LIN {X -0.096,Y -433.923,Z 789.927,A 0.000,B 0.000,C 90.000,E1 202.950} C_DIS
LIN {X -0.182,Y -428.835,Z 789.913,A 0.000,B 0.000,C 90.000,E1 200.301} C_DIS
LIN {X -0.108,Y -424.366,Z 789.900,A 0.000,B 0.000,C 90.000,E1 197.946} C_DIS
LIN {X 0.063,Y -420.410,Z 789.888,A 0.000,B 0.000,C 90.000,E1 195.898} C_DIS
LIN {X 0.140,Y -414.585,Z 789.871,A 0.000,B 0.000,C 90.000,E1 192.827} C_DIS
LIN {X -0.010,Y -412.023,Z 789.864,A 0.000,B 0.000,C 90.000,E1 191.478} C_DIS
LIN {X -0.175,Y -407.184,Z 789.849,A 0.000,B 0.000,C 90.000,E1 188.746} C_DIS
LIN {X -0.117,Y -404.851,Z 789.841,A 0.000,B 0.000,C 90.000,E1 187.352} C_DIS
LIN {X 0.135,Y -400.530,Z 789.827,A 0.000,B 0.000,C 90.000,E1 184.878} C_DIS
LIN {X -0.196,Y -393.502,Z 789.800,A 0.000,B 0.000,C 90.000,E1 180.000} C_DIS
LIN {X -0.078,Y -390.107,Z 789.782,A 0.000,B 0.000,C 90.000,E1 176.788} C_DIS
LIN {X -0.091,Y -388.317,Z 789.772,A 0.000,B 0.000,C 90.000,E1 175.008} C_DIS
LIN {X 0.135,Y -385.736,Z 789.758,A 0.000,B 0.000,C 90.000,E1 172.470} C_DIS
LIN {X 0.177,Y -384.408,Z 789.750,A 0.000,B 0.000,C 90.000,E1 171.027} C_DIS
LIN {X -0.013,Y -381.815,Z 789.732,A 0.000,B 0.000,C 90.000,E1 167.813} C_DIS
LIN {X -0.019,Y -380.151,Z 789.718,A 0.000,B 0.000,C 90.000,E1 165.283} C_DIS
LIN {X 0.113,Y -378.893,Z 789.704,A 0.000,B 0.000,C 90.000,E1 162.725} C_DIS
LIN {X 0.069,Y -377.980,Z 789.690,A 0.000,B 0.000,C 90.000,E1 160.188} C_DIS
LIN {X -0.095,Y -377.646,Z 789.676,A 0.000,B 0.000,C 90.000,E1 157.667} C_DIS
LIN {X -0.228,Y -379.156,Z 789.646,A 0.000,B 0.000,C 90.000,E1 152.231} C_DIS
LIN {X 0.139,Y -380.892,Z 789.633,A 0.000,B 0.000,C 90.000,E1 149.999} C_DIS
LIN {X 0.074,Y -383.379,Z 789.623,A 0.000,B 0.000,C 90.000,E1 148.201} C_DIS
LIN {X -0.076,Y -384.604,Z 789.619,A 0.000,B 0.000,C 90.000,E1 147.502} C_DIS
LIN {X 0.144,Y -388.645,Z 789.609,A 0.000,B 0.000,C 90.000,E1 145.674} C_DIS
LIN {X 0.039,Y -390.655,Z 789.606,A 0.000,B 0.000,C 90.000,E1 144.975} C_DIS
LIN {X -0.048,Y -393.112,Z 789.602,A 0.000,B 0.000,C 90.000,E1 144.276} C_DIS
LIN {X 0.119,Y -396.079,Z 789.598,A 0.000,B 0.000,C 90.000,E1 143.543} C_DIS
LIN {X 0.038,Y -400.422,Z 789.593,A 0.000,B 0.000,C 90.000,E1 142.718} C_DIS
LIN {X 0.118,Y -403.485,Z 789.590,A 0.000,B 0.000,C 90.000,E1 142.190} C_DIS
LIN {X 0.232,Y -407.862,Z 789.587,A 0.000,B 0.000,C 90.000,E1 141.537} C_DIS
LIN {X 0.073,Y -425.471,Z 789.574,A 0.000,B 0.000,C 90.000,E1 139.380} C_DIS
LIN {X -0.229,Y -441.850,Z 789.564,A 0.000,B 0.000,C 90.000,E1 137.472} C_DIS
LIN {X -0.276,Y -452.614,Z 789.557,A 0.000,B 0.000,C 90.000,E1 136.215} C_DIS
LIN {X -0.051,Y -461.582,Z 789.550,A 0.000,B 0.000,C 90.000,E1 135.081} C_DIS
LIN {X 0.114,Y -468.893,Z 789.545,A 0.000,B 0.000,C 90.000,E1 134.109} C_DIS
LIN {X 0.245,Y -478.125,Z 789.538,A 0.000,B 0.000,C 90.000,E1 132.852} C_DIS
LIN {X -0.339,Y -485.771,Z 789.532,A 0.000,B 0.000,C 90.000,E1 131.838} C_DIS
LIN {X -0.279,Y -490.960,Z 789.528,A 0.000,B 0.000,C 90.000,E1 131.067} C_DIS
LIN {X 0.220,Y -499.566,Z 789.520,A 0.000,B 0.000,C 90.000,E1 129.644} C_DIS
LIN {X 0.167,Y -505.023,Z 789.515,A 0.000,B 0.000,C 90.000,E1 128.749} C_DIS
LIN {X -0.143,Y -510.126,Z 789.510,A 0.000,B 0.000,C 90.000,E1 127.890} C_DIS
LIN {X -0.009,Y -513.345,Z 789.507,A 0.000,B 0.000,C 90.000,E1 127.282} C_DIS
LIN {X -0.063,Y -520.174,Z 789.500,A 0.000,B 0.000,C 90.000,E1 125.964} C_DIS
LIN {X -0.253,Y -525.997,Z 789.493,A 0.000,B 0.000,C 90.000,E1 124.818} C_DIS
LIN {X 0.086,Y -529.747,Z 789.489,A 0.000,B 0.000,C 90.000,E1 123.913} C_DIS
LIN {X 0.176,Y -533.294,Z 789.484,A 0.000,B 0.000,C 90.000,E1 123.038} C_DIS
LIN {X -0.148,Y -536.722,Z 789.479,A 0.000,B 0.000,C 90.000,E1 122.212} C_DIS
LIN {X 0.021,Y -541.048,Z 789.473,A 0.000,B 0.000,C 90.000,E1 121.052} C_DIS
LIN {X -0.044,Y -544.102,Z 789.468,A 0.000,B 0.000,C 90.000,E1 120.207} C_DIS
LIN {X 0.200,Y -546.907,Z 789.463,A 0.000,B 0.000,C 90.000,E1 119.333} C_DIS
LIN {X -0.036,Y -550.394,Z 789.457,A 0.000,B 0.000,C 90.000,E1 118.231} C_DIS
LIN {X 0.008,Y -552.853,Z 789.452,A 0.000,B 0.000,C 90.000,E1 117.385} C_DIS
LIN {X 0.073,Y -554.977,Z 789.448,A 0.000,B 0.000,C 90.000,E1 116.539} C_DIS
LIN {X -0.087,Y -556.744,Z 789.443,A 0.000,B 0.000,C 90.000,E1 115.720} C_DIS
LIN {X -0.225,Y -558.214,Z 789.438,A 0.000,B 0.000,C 90.000,E1 114.899} C_DIS
LIN {X 0.164,Y -559.424,Z 789.434,A 0.000,B 0.000,C 90.000,E1 114.027} C_DIS
LIN {X 0.157,Y -560.882,Z 789.426,A 0.000,B 0.000,C 90.000,E1 112.642} C_DIS
LIN {X -0.047,Y -562.323,Z 789.418,A 0.000,B 0.000,C 90.000,E1 111.280} C_DIS
LIN {X 0.098,Y -563.529,Z 789.411,A 0.000,B 0.000,C 90.000,E1 109.885} C_DIS
LIN {X -0.262,Y -564.477,Z 789.403,A 0.000,B 0.000,C 90.000,E1 108.544} C_DIS
LIN {X 0.071,Y -565.546,Z 789.394,A 0.000,B 0.000,C 90.000,E1 106.858} C_DIS
LIN {X 0.053,Y -566.949,Z 789.382,A 0.000,B 0.000,C 90.000,E1 104.662} C_DIS
LIN {X -0.061,Y -568.582,Z 789.369,A 0.000,B 0.000,C 90.000,E1 102.479} C_DIS
LIN {X 0.109,Y -570.137,Z 789.359,A 0.000,B 0.000,C 90.000,E1 100.546} C_DIS
LIN {X 0.202,Y -571.656,Z 789.348,A 0.000,B 0.000,C 90.000,E1 98.624} C_DIS
LIN {X -0.147,Y -572.602,Z 789.341,A 0.000,B 0.000,C 90.000,E1 97.296} C_DIS
LIN {X 0.217,Y -573.687,Z 789.331,A 0.000,B 0.000,C 90.000,E1 95.625} C_DIS
LIN {X 0.166,Y -574.755,Z 789.321,A 0.000,B 0.000,C 90.000,E1 93.726} C_DIS
LIN {X -0.229,Y -575.442,Z 789.313,A 0.000,B 0.000,C 90.000,E1 92.407} C_DIS
LIN {X -0.037,Y -575.998,Z 789.306,A 0.000,B 0.000,C 90.000,E1 91.031} C_DIS
LIN {X -0.270,Y -576.652,Z 789.297,A 0.000,B 0.000,C 90.000,E1 89.427} C_DIS
LIN {X 0.193,Y -576.956,Z 789.292,A 0.000,B 0.000,C 90.000,E1 88.568} C_DIS
LIN {X -0.013,Y -577.454,Z 789.283,A 0.000,B 0.000,C 90.000,E1 86.963} C_DIS
LIN {X 0.245,Y -577.727,Z 789.276,A 0.000,B 0.000,C 90.000,E1 85.584} C_DIS
LIN {X 0.144,Y -578.060,Z 789.267,A 0.000,B 0.000,C 90.000,E1 83.970} C_DIS
LIN {X 0.050,Y -578.363,Z 789.258,A 0.000,B 0.000,C 90.000,E1 82.356} C_DIS
LIN {X 0.030,Y -578.620,Z 789.249,A 0.000,B 0.000,C 90.000,E1 80.735} C_DIS
LIN {X 0.107,Y -578.803,Z 789.240,A 0.000,B 0.000,C 90.000,E1 79.106} C_DIS
LIN {X 0.079,Y -578.817,Z 789.232,A 0.000,B 0.000,C 90.000,E1 77.757} C_DIS
LIN {X 0.051,Y -578.707,Z 789.225,A 0.000,B 0.000,C 90.000,E1 76.408} C_DIS
LIN {X -0.061,Y -578.550,Z 789.219,A 0.000,B 0.000,C 90.000,E1 75.338} C_DIS
LIN {X -0.099,Y -578.141,Z 789.208,A 0.000,B 0.000,C 90.000,E1 73.449} C_DIS
LIN {X 0.144,Y -577.788,Z 789.201,A 0.000,B 0.000,C 90.000,E1 72.072} C_DIS
LIN {X -0.007,Y -577.504,Z 789.196,A 0.000,B 0.000,C 90.000,E1 71.275} C_DIS
LIN {X 0.046,Y -576.855,Z 789.187,A 0.000,B 0.000,C 90.000,E1 69.645} C_DIS
LIN {X -0.050,Y -576.024,Z 789.178,A 0.000,B 0.000,C 90.000,E1 68.028} C_DIS
LIN {X 0.008,Y -575.252,Z 789.170,A 0.000,B 0.000,C 90.000,E1 66.666} C_DIS
LIN {X 0.039,Y -574.268,Z 789.163,A 0.000,B 0.000,C 90.000,E1 65.305} C_DIS
LIN {X 0.172,Y -573.461,Z 789.157,A 0.000,B 0.000,C 90.000,E1 64.204} C_DIS
LIN {X -0.113,Y -572.147,Z 789.149,A 0.000,B 0.000,C 90.000,E1 62.871} C_DIS
LIN {X 0.001,Y -570.894,Z 789.143,A 0.000,B 0.000,C 90.000,E1 61.769} C_DIS
LIN {X -0.081,Y -568.995,Z 789.136,A 0.000,B 0.000,C 90.000,E1 60.411} C_DIS
LIN {X -0.047,Y -567.718,Z 789.131,A 0.000,B 0.000,C 90.000,E1 59.587} C_DIS
LIN {X -0.013,Y -565.741,Z 789.125,A 0.000,B 0.000,C 90.000,E1 58.486} C_DIS
LIN {X -0.003,Y -564.109,Z 789.120,A 0.000,B 0.000,C 90.000,E1 57.661} C_DIS
LIN {X -0.005,Y -562.277,Z 789.116,A 0.000,B 0.000,C 90.000,E1 56.834} C_DIS
LIN {X -0.025,Y -560.239,Z 789.111,A 0.000,B 0.000,C 90.000,E1 56.008} C_DIS
LIN {X -0.067,Y -557.981,Z 789.107,A 0.000,B 0.000,C 90.000,E1 55.182} C_DIS
LIN {X -0.137,Y -555.469,Z 789.102,A 0.000,B 0.000,C 90.000,E1 54.356} C_DIS
LIN {X 0.016,Y -553.739,Z 789.099,A 0.000,B 0.000,C 90.000,E1 53.783} C_DIS
LIN {X 0.222,Y -550.798,Z 789.094,A 0.000,B 0.000,C 90.000,E1 52.924} C_DIS
LIN {X -0.038,Y -547.508,Z 789.090,A 0.000,B 0.000,C 90.000,E1 52.110} C_DIS
LIN {X -0.091,Y -544.513,Z 789.086,A 0.000,B 0.000,C 90.000,E1 51.412} C_DIS
LIN {X -0.258,Y -541.278,Z 789.082,A 0.000,B 0.000,C 90.000,E1 50.723} C_DIS
LIN {X 0.130,Y -538.423,Z 789.079,A 0.000,B 0.000,C 90.000,E1 50.114} C_DIS
LIN {X 0.321,Y -534.466,Z 789.075,A 0.000,B 0.000,C 90.000,E1 49.380} C_DIS
LIN {X -0.052,Y -531.062,Z 789.071,A 0.000,B 0.000,C 90.000,E1 48.852} C_DIS
LIN {X 0.254,Y -527.176,Z 789.068,A 0.000,B 0.000,C 90.000,E1 48.243} C_DIS
LIN {X -0.212,Y -522.843,Z 789.065,A 0.000,B 0.000,C 90.000,E1 47.715} C_DIS
LIN {X -0.215,Y -518.175,Z 789.062,A 0.000,B 0.000,C 90.000,E1 47.148} C_DIS
LIN {X -0.127,Y -514.389,Z 789.059,A 0.000,B 0.000,C 90.000,E1 46.701} C_DIS
LIN {X -0.219,Y -508.950,Z 789.056,A 0.000,B 0.000,C 90.000,E1 46.134} C_DIS
LIN {X -0.306,Y -504.703,Z 789.054,A 0.000,B 0.000,C 90.000,E1 45.729} C_DIS
LIN {X -0.045,Y -497.382,Z 789.050,A 0.000,B 0.000,C 90.000,E1 45.040} C_DIS
LIN {X 0.203,Y -494.493,Z 789.049,A 0.000,B 0.000,C 90.000,E1 44.757} C_DIS
LIN {X -0.244,Y -486.605,Z 789.045,A 0.000,B 0.000,C 90.000,E1 44.190} C_DIS
LIN {X -0.048,Y -478.786,Z 789.042,A 0.000,B 0.000,C 90.000,E1 43.581} C_DIS
LIN {X -0.066,Y -465.969,Z 789.037,A 0.000,B 0.000,C 90.000,E1 42.690} C_DIS
LIN {X -0.267,Y -452.980,Z 789.032,A 0.000,B 0.000,C 90.000,E1 41.838} C_DIS
LIN {X -0.082,Y -427.596,Z 789.022,A 0.000,B 0.000,C 90.000,E1 40.011} C_DIS
LIN {X -0.153,Y -415.102,Z 789.017,A 0.000,B 0.000,C 90.000,E1 39.036} C_DIS
LIN {X -0.015,Y -409.294,Z 789.014,A 0.000,B 0.000,C 90.000,E1 38.508} C_DIS
LIN {X -0.120,Y -404.958,Z 789.012,A 0.000,B 0.000,C 90.000,E1 38.096} C_DIS
LIN {X -0.153,Y -404.943,Z 789.012,A 0.000,B 0.000,C 90.000,E1 38.096} C_DIS
LIN {X -0.008,Y -396.699,Z 788.988,A 0.000,B 0.000,C 90.000,E1 33.785} C_DIS
LIN {X 0.077,Y -395.965,Z 788.985,A 0.000,B 0.000,C 90.000,E1 33.245} C_DIS
LIN {X 0.145,Y -396.699,Z 788.970,A 0.000,B 0.000,C 90.000,E1 30.590} C_DIS
LIN {X 0.174,Y -398.039,Z 788.954,A 0.000,B 0.000,C 90.000,E1 27.769} C_DIS
LIN {X -0.003,Y -399.440,Z 788.941,A 0.000,B 0.000,C 90.000,E1 25.335} C_DIS
LIN {X 0.178,Y -400.863,Z 788.929,A 0.000,B 0.000,C 90.000,E1 23.206} C_DIS
LIN {X 0.143,Y -403.490,Z 788.912,A 0.000,B 0.000,C 90.000,E1 20.066} C_DIS
LIN {X 0.024,Y -407.875,Z 788.890,A 0.000,B 0.000,C 90.000,E1 16.260} C_DIS
LIN {X -0.123,Y -412.436,Z 788.873,A 0.000,B 0.000,C 90.000,E1 13.175} C_DIS
LIN {X -0.165,Y -416.506,Z 788.860,A 0.000,B 0.000,C 90.000,E1 10.782} C_DIS
LIN {X -0.227,Y -420.048,Z 788.848,A 0.000,B 0.000,C 90.000,E1 8.746} C_DIS
LIN {X 0.150,Y -423.655,Z 788.837,A 0.000,B 0.000,C 90.000,E1 6.663} C_DIS
LIN {X 0.189,Y -427.918,Z 788.824,A 0.000,B 0.000,C 90.000,E1 4.302} C_DIS
LIN {X 0.210,Y -431.687,Z 788.813,A 0.000,B 0.000,C 90.000,E1 2.293} C_DIS
LIN {X 0.165,Y -436.770,Z 788.799,A 0.000,B 0.000,C 90.000,E1 359.771} C_DIS
LIN {X 0.176,Y -442.483,Z 788.784,A 0.000,B 0.000,C 90.000,E1 357.135} C_DIS
LIN {X -0.176,Y -447.843,Z 788.772,A 0.000,B 0.000,C 90.000,E1 354.894} C_DIS
LIN {X 0.104,Y -453.252,Z 788.759,A 0.000,B 0.000,C 90.000,E1 352.591} C_DIS
LIN {X 0.199,Y -457.058,Z 788.750,A 0.000,B 0.000,C 90.000,E1 350.971} C_DIS
LIN {X -0.188,Y -463.295,Z 788.736,A 0.000,B 0.000,C 90.000,E1 348.465} C_DIS
LIN {X -0.048,Y -465.363,Z 788.732,A 0.000,B 0.000,C 90.000,E1 347.813} C_DIS
LIN {X 0.209,Y -466.568,Z 788.731,A 0.000,B 0.000,C 90.000,E1 347.465} C_DIS
LIN {X -0.121,Y -468.502,Z 788.728,A 0.000,B 0.000,C 90.000,E1 347.117} C_DIS
LIN {X 0.118,Y -471.921,Z 788.726,A 0.000,B 0.000,C 90.000,E1 346.589} C_DIS
LIN {X 0.192,Y -476.026,Z 788.723,A 0.000,B 0.000,C 90.000,E1 346.117} C_DIS
LIN {X 0.085,Y -481.163,Z 788.720,A 0.000,B 0.000,C 90.000,E1 345.644} C_DIS
LIN {X 0.074,Y -492.813,Z 788.715,A 0.000,B 0.000,C 90.000,E1 344.755} C_DIS
LIN {X -0.016,Y -511.779,Z 788.708,A 0.000,B 0.000,C 90.000,E1 343.449} C_DIS
LIN {X -0.203,Y -530.426,Z 788.701,A 0.000,B 0.000,C 90.000,E1 342.236} C_DIS
LIN {X 0.002,Y -538.135,Z 788.698,A 0.000,B 0.000,C 90.000,E1 341.692} C_DIS
LIN {X -0.207,Y -548.725,Z 788.694,A 0.000,B 0.000,C 90.000,E1 340.967} C_DIS
LIN {X 0.155,Y -555.920,Z 788.691,A 0.000,B 0.000,C 90.000,E1 340.369} C_DIS
LIN {X 0.240,Y -561.405,Z 788.688,A 0.000,B 0.000,C 90.000,E1 339.880} C_DIS
LIN {X 0.036,Y -566.649,Z 788.686,A 0.000,B 0.000,C 90.000,E1 339.390} C_DIS
LIN {X 0.117,Y -571.621,Z 788.683,A 0.000,B 0.000,C 90.000,E1 338.847} C_DIS
LIN {X 0.246,Y -577.291,Z 788.679,A 0.000,B 0.000,C 90.000,E1 338.156} C_DIS
LIN {X 0.113,Y -583.671,Z 788.674,A 0.000,B 0.000,C 90.000,E1 337.358} C_DIS
LIN {X 0.330,Y -588.579,Z 788.671,A 0.000,B 0.000,C 90.000,E1 336.666} C_DIS
LIN {X 0.206,Y -595.966,Z 788.665,A 0.000,B 0.000,C 90.000,E1 335.613} C_DIS
LIN {X -0.085,Y -602.129,Z 788.660,A 0.000,B 0.000,C 90.000,E1 334.717} C_DIS
LIN {X 0.220,Y -608.704,Z 788.654,A 0.000,B 0.000,C 90.000,E1 333.640} C_DIS
LIN {X 0.067,Y -614.861,Z 788.648,A 0.000,B 0.000,C 90.000,E1 332.615} C_DIS
LIN {X -0.004,Y -620.008,Z 788.643,A 0.000,B 0.000,C 90.000,E1 331.719} C_DIS
LIN {X -0.264,Y -625.689,Z 788.637,A 0.000,B 0.000,C 90.000,E1 330.717} C_DIS
LIN {X 0.103,Y -631.070,Z 788.632,A 0.000,B 0.000,C 90.000,E1 329.665} C_DIS
LIN {X 0.016,Y -636.701,Z 788.625,A 0.000,B 0.000,C 90.000,E1 328.535} C_DIS
LIN {X -0.071,Y -640.189,Z 788.621,A 0.000,B 0.000,C 90.000,E1 327.788} C_DIS
LIN {X -0.073,Y -644.643,Z 788.615,A 0.000,B 0.000,C 90.000,E1 326.786} C_DIS
LIN {X -0.147,Y -646.699,Z 788.613,A 0.000,B 0.000,C 90.000,E1 326.294} C_DIS
LIN {X -0.246,Y -650.752,Z 788.607,A 0.000,B 0.000,C 90.000,E1 325.308} C_DIS
LIN {X 0.245,Y -654.480,Z 788.602,A 0.000,B 0.000,C 90.000,E1 324.276} C_DIS
LIN {X -0.280,Y -658.009,Z 788.596,A 0.000,B 0.000,C 90.000,E1 323.336} C_DIS
LIN {X -0.278,Y -662.012,Z 788.589,A 0.000,B 0.000,C 90.000,E1 322.110} C_DIS
LIN {X -0.214,Y -665.758,Z 788.583,A 0.000,B 0.000,C 90.000,E1 320.884} C_DIS
LIN {X -0.185,Y -669.185,Z 788.576,A 0.000,B 0.000,C 90.000,E1 319.666} C_DIS
LIN {X -0.102,Y -671.762,Z 788.570,A 0.000,B 0.000,C 90.000,E1 318.690} C_DIS
LIN {X 0.027,Y -674.793,Z 788.564,A 0.000,B 0.000,C 90.000,E1 317.472} C_DIS
LIN {X -0.298,Y -677.372,Z 788.557,A 0.000,B 0.000,C 90.000,E1 316.296} C_DIS
LIN {X -0.026,Y -680.472,Z 788.548,A 0.000,B 0.000,C 90.000,E1 314.595} C_DIS
LIN {X 0.209,Y -682.391,Z 788.541,A 0.000,B 0.000,C 90.000,E1 313.380} C_DIS
LIN {X -0.001,Y -684.231,Z 788.535,A 0.000,B 0.000,C 90.000,E1 312.204} C_DIS
LIN {X 0.327,Y -685.870,Z 788.528,A 0.000,B 0.000,C 90.000,E1 310.987} C_DIS
LIN {X 0.239,Y -687.268,Z 788.521,A 0.000,B 0.000,C 90.000,E1 309.806} C_DIS
LIN {X 0.180,Y -688.502,Z 788.515,A 0.000,B 0.000,C 90.000,E1 308.624} C_DIS
LIN {X -0.186,Y -690.165,Z 788.505,A 0.000,B 0.000,C 90.000,E1 306.996} C_DIS
LIN {X -0.438,Y -691.394,Z 788.498,A 0.000,B 0.000,C 90.000,E1 305.598} C_DIS
LIN {X -0.302,Y -692.289,Z 788.491,A 0.000,B 0.000,C 90.000,E1 304.405} C_DIS
LIN {X -0.290,Y -693.500,Z 788.482,A 0.000,B 0.000,C 90.000,E1 302.752} C_DIS
LIN {X -0.032,Y -694.830,Z 788.473,A 0.000,B 0.000,C 90.000,E1 301.082} C_DIS
LIN {X 0.111,Y -695.492,Z 788.467,A 0.000,B 0.000,C 90.000,E1 300.129} C_DIS
LIN {X -0.197,Y -696.213,Z 788.460,A 0.000,B 0.000,C 90.000,E1 298.743} C_DIS
LIN {X 0.215,Y -696.715,Z 788.454,A 0.000,B 0.000,C 90.000,E1 297.769} C_DIS
LIN {X 0.216,Y -697.495,Z 788.447,A 0.000,B 0.000,C 90.000,E1 296.360} C_DIS
LIN {X 0.232,Y -698.424,Z 788.439,A 0.000,B 0.000,C 90.000,E1 294.951} C_DIS
LIN {X -0.169,Y -698.589,Z 788.436,A 0.000,B 0.000,C 90.000,E1 294.515} C_DIS
LIN {X 0.094,Y -698.627,Z 788.435,A 0.000,B 0.000,C 90.000,E1 294.259} C_DIS
LIN {X 0.072,Y -698.429,Z 788.434,A 0.000,B 0.000,C 90.000,E1 294.027} C_DIS
LIN {X -0.042,Y -697.521,Z 788.431,A 0.000,B 0.000,C 90.000,E1 293.567} C_DIS
LIN {X -0.060,Y -696.532,Z 788.430,A 0.000,B 0.000,C 90.000,E1 293.334} C_DIS
LIN {X 0.321,Y -693.962,Z 788.428,A 0.000,B 0.000,C 90.000,E1 292.950} C_DIS
LIN {X -0.341,Y -692.008,Z 788.426,A 0.000,B 0.000,C 90.000,E1 292.770} C_DIS
LIN {X -0.220,Y -690.406,Z 788.426,A 0.000,B 0.000,C 90.000,E1 292.642} C_DIS
LIN {X 0.151,Y -686.156,Z 788.425,A 0.000,B 0.000,C 90.000,E1 292.408} C_DIS
LIN {X -0.086,Y -682.793,Z 788.424,A 0.000,B 0.000,C 90.000,E1 292.280} C_DIS
LIN {X -0.037,Y -680.715,Z 788.423,A 0.000,B 0.000,C 90.000,E1 292.206} C_DIS
LIN {X 0.087,Y -674.471,Z 788.422,A 0.000,B 0.000,C 90.000,E1 292.025} C_DIS
LIN {X -0.131,Y -669.195,Z 788.422,A 0.000,B 0.000,C 90.000,E1 291.950} C_DIS
LIN {X -0.150,Y -651.406,Z 788.420,A 0.000,B 0.000,C 90.000,E1 291.663} C_DIS
LIN {X -0.111,Y -634.211,Z 788.419,A 0.000,B 0.000,C 90.000,E1 291.334} C_DIS
LIN {X -0.087,Y -613.288,Z 788.416,A 0.000,B 0.000,C 90.000,E1 290.865} C_DIS
LIN {X -0.083,Y -596.538,Z 788.414,A 0.000,B 0.000,C 90.000,E1 290.429} C_DIS
LIN {X 0.072,Y -586.447,Z 788.412,A 0.000,B 0.000,C 90.000,E1 290.120} C_DIS
LIN {X -0.132,Y -576.325,Z 788.410,A 0.000,B 0.000,C 90.000,E1 289.812} C_DIS
LIN {X -0.045,Y -569.864,Z 788.409,A 0.000,B 0.000,C 90.000,E1 289.577} C_DIS
LIN {X 0.055,Y -564.207,Z 788.407,A 0.000,B 0.000,C 90.000,E1 289.322} C_DIS
LIN {X 0.105,Y -562.387,Z 788.407,A 0.000,B 0.000,C 90.000,E1 289.214} C_DIS
LIN {X -0.020,Y -558.873,Z 788.405,A 0.000,B 0.000,C 90.000,E1 288.960} C_DIS
LIN {X -0.139,Y -557.615,Z 788.404,A 0.000,B 0.000,C 90.000,E1 288.779} C_DIS
LIN {X 0.273,Y -556.882,Z 788.404,A 0.000,B 0.000,C 90.000,E1 288.598} C_DIS
LIN {X 0.139,Y -555.816,Z 788.402,A 0.000,B 0.000,C 90.000,E1 288.308} C_DIS
LIN {X -0.011,Y -555.004,Z 788.400,A 0.000,B 0.000,C 90.000,E1 287.946} C_DIS
LIN {X -0.143,Y -554.325,Z 788.397,A 0.000,B 0.000,C 90.000,E1 287.402} C_DIS
LIN {X -0.156,Y -552.737,Z 788.376,A 0.000,B 0.000,C 90.000,E1 283.772} C_DIS
LIN {X 0.147,Y -552.218,Z 788.367,A 0.000,B 0.000,C 90.000,E1 282.063} C_DIS
LIN {X -0.210,Y -551.653,Z 788.356,A 0.000,B 0.000,C 90.000,E1 280.141} C_DIS
LIN {X 0.104,Y -551.022,Z 788.342,A 0.000,B 0.000,C 90.000,E1 277.587} C_DIS
LIN {X -0.085,Y -550.591,Z 788.336,A 0.000,B 0.000,C 90.000,E1 276.486} C_DIS
LIN {X -0.213,Y -549.742,Z 788.327,A 0.000,B 0.000,C 90.000,E1 274.816} C_DIS
LIN {X 0.062,Y -548.791,Z 788.319,A 0.000,B 0.000,C 90.000,E1 273.383} C_DIS
LIN {X -0.104,Y -547.554,Z 788.308,A 0.000,B 0.000,C 90.000,E1 271.432} C_DIS
LIN {X 0.170,Y -546.472,Z 788.299,A 0.000,B 0.000,C 90.000,E1 269.714} C_DIS
LIN {X -0.168,Y -545.463,Z 788.291,A 0.000,B 0.000,C 90.000,E1 268.339} C_DIS
LIN {X 0.094,Y -544.340,Z 788.281,A 0.000,B 0.000,C 90.000,E1 266.617} C_DIS
LIN {X -0.272,Y -543.516,Z 788.273,A 0.000,B 0.000,C 90.000,E1 265.241} C_DIS
LIN {X -0.009,Y -542.383,Z 788.264,A 0.000,B 0.000,C 90.000,E1 263.514} C_DIS
LIN {X 0.293,Y -541.219,Z 788.256,A 0.000,B 0.000,C 90.000,E1 262.064} C_DIS
LIN {X 0.109,Y -539.568,Z 788.245,A 0.000,B 0.000,C 90.000,E1 260.095} C_DIS
LIN {X -0.237,Y -538.504,Z 788.239,A 0.000,B 0.000,C 90.000,E1 258.993} C_DIS
LIN {X 0.266,Y -536.864,Z 788.229,A 0.000,B 0.000,C 90.000,E1 257.229} C_DIS
LIN {X -0.019,Y -535.770,Z 788.223,A 0.000,B 0.000,C 90.000,E1 256.117} C_DIS
LIN {X 0.081,Y -533.559,Z 788.212,A 0.000,B 0.000,C 90.000,E1 254.102} C_DIS
LIN {X 0.239,Y -531.630,Z 788.202,A 0.000,B 0.000,C 90.000,E1 252.362} C_DIS
LIN {X -0.166,Y -529.904,Z 788.194,A 0.000,B 0.000,C 90.000,E1 250.967} C_DIS
LIN {X 0.076,Y -527.478,Z 788.185,A 0.000,B 0.000,C 90.000,E1 249.209} C_DIS
LIN {X -0.220,Y -525.416,Z 788.177,A 0.000,B 0.000,C 90.000,E1 247.794} C_DIS
LIN {X -0.035,Y -523.614,Z 788.170,A 0.000,B 0.000,C 90.000,E1 246.613} C_DIS
LIN {X 0.017,Y -521.396,Z 788.162,A 0.000,B 0.000,C 90.000,E1 245.153} C_DIS
LIN {X 0.035,Y -519.030,Z 788.154,A 0.000,B 0.000,C 90.000,E1 243.691} C_DIS
LIN {X -0.124,Y -517.079,Z 788.147,A 0.000,B 0.000,C 90.000,E1 242.538} C_DIS
LIN {X 0.023,Y -515.509,Z 788.143,A 0.000,B 0.000,C 90.000,E1 241.641} C_DIS
LIN {X -0.298,Y -512.749,Z 788.134,A 0.000,B 0.000,C 90.000,E1 240.205} C_DIS
LIN {X 0.285,Y -509.978,Z 788.126,A 0.000,B 0.000,C 90.000,E1 238.663} C_DIS
LIN {X 0.004,Y -506.328,Z 788.116,A 0.000,B 0.000,C 90.000,E1 236.914} C_DIS
LIN {X 0.109,Y -504.427,Z 788.111,A 0.000,B 0.000,C 90.000,E1 236.008} C_DIS
LIN {X 0.083,Y -501.692,Z 788.105,A 0.000,B 0.000,C 90.000,E1 234.815} C_DIS
LIN {X 0.139,Y -499.536,Z 788.100,A 0.000,B 0.000,C 90.000,E1 233.909} C_DIS
LIN {X -0.100,Y -495.775,Z 788.091,A 0.000,B 0.000,C 90.000,E1 232.431} C_DIS
LIN {X 0.199,Y -490.501,Z 788.079,A 0.000,B 0.000,C 90.000,E1 230.275} C_DIS
LIN {X -0.046,Y -484.219,Z 788.064,A 0.000,B 0.000,C 90.000,E1 227.553} C_DIS
LIN {X -0.248,Y -480.260,Z 788.054,A 0.000,B 0.000,C 90.000,E1 225.729} C_DIS
LIN {X -0.315,Y -476.825,Z 788.045,A 0.000,B 0.000,C 90.000,E1 224.190} C_DIS
LIN {X -0.108,Y -473.429,Z 788.037,A 0.000,B 0.000,C 90.000,E1 222.609} C_DIS
LIN {X -0.011,Y -468.094,Z 788.023,A 0.000,B 0.000,C 90.000,E1 220.092} C_DIS
LIN {X 0.175,Y -464.060,Z 788.012,A 0.000,B 0.000,C 90.000,E1 218.177} C_DIS
LIN {X -0.159,Y -461.517,Z 788.005,A 0.000,B 0.000,C 90.000,E1 216.950} C_DIS
LIN {X 0.066,Y -456.774,Z 787.993,A 0.000,B 0.000,C 90.000,E1 214.692} C_DIS
LIN {X 0.181,Y -452.912,Z 787.982,A 0.000,B 0.000,C 90.000,E1 212.752} C_DIS
LIN {X -0.199,Y -448.467,Z 787.970,A 0.000,B 0.000,C 90.000,E1 210.541} C_DIS
LIN {X 0.015,Y -444.689,Z 787.959,A 0.000,B 0.000,C 90.000,E1 208.565} C_DIS
LIN {X 0.079,Y -441.606,Z 787.950,A 0.000,B 0.000,C 90.000,E1 206.924} C_DIS
LIN {X 0.075,Y -438.468,Z 787.941,A 0.000,B 0.000,C 90.000,E1 205.283} C_DIS
LIN {X -0.154,Y -434.747,Z 787.930,A 0.000,B 0.000,C 90.000,E1 203.334} C_DIS
LIN {X -0.053,Y -429.614,Z 787.915,A 0.000,B 0.000,C 90.000,E1 200.663} C_DIS
LIN {X -0.022,Y -427.031,Z 787.907,A 0.000,B 0.000,C 90.000,E1 199.322} C_DIS
LIN {X 0.023,Y -423.876,Z 787.898,A 0.000,B 0.000,C 90.000,E1 197.638} C_DIS
LIN {X -0.112,Y -420.584,Z 787.889,A 0.000,B 0.000,C 90.000,E1 195.969} C_DIS
LIN {X 0.081,Y -414.772,Z 787.872,A 0.000,B 0.000,C 90.000,E1 192.883} C_DIS
LIN {X -0.106,Y -412.860,Z 787.866,A 0.000,B 0.000,C 90.000,E1 191.883} C_DIS
LIN {X -0.196,Y -406.222,Z 787.845,A 0.000,B 0.000,C 90.000,E1 188.106} C_DIS
LIN {X -0.209,Y -403.792,Z 787.837,A 0.000,B 0.000,C 90.000,E1 186.720} C_DIS
LIN {X 0.070,Y -400.201,Z 787.826,A 0.000,B 0.000,C 90.000,E1 184.588} C_DIS
LIN {X 0.160,Y -393.706,Z 787.800,A 0.000,B 0.000,C 90.000,E1 180.000} C_DIS
LIN {X -0.108,Y -390.325,Z 787.782,A 0.000,B 0.000,C 90.000,E1 176.846} C_DIS
LIN {X -0.116,Y -388.547,Z 787.773,A 0.000,B 0.000,C 90.000,E1 175.065} C_DIS
LIN {X -0.129,Y -386.637,Z 787.763,A 0.000,B 0.000,C 90.000,E1 173.280} C_DIS
LIN {X -0.141,Y -385.015,Z 787.753,A 0.000,B 0.000,C 90.000,E1 171.489} C_DIS
LIN {X -0.005,Y -382.332,Z 787.735,A 0.000,B 0.000,C 90.000,E1 168.229} C_DIS
LIN {X 0.100,Y -381.303,Z 787.727,A 0.000,B 0.000,C 90.000,E1 166.769} C_DIS
LIN {X -0.003,Y -380.492,Z 787.719,A 0.000,B 0.000,C 90.000,E1 165.338} C_DIS
LIN {X 0.141,Y -379.058,Z 787.702,A 0.000,B 0.000,C 90.000,E1 162.417} C_DIS
LIN {X 0.113,Y -378.334,Z 787.690,A 0.000,B 0.000,C 90.000,E1 160.242} C_DIS
LIN {X -0.050,Y -377.905,Z 787.674,A 0.000,B 0.000,C 90.000,E1 157.358} C_DIS
LIN {X 0.098,Y -380.351,Z 787.638,A 0.000,B 0.000,C 90.000,E1 150.795} C_DIS
LIN {X -0.135,Y -381.354,Z 787.632,A 0.000,B 0.000,C 90.000,E1 149.744} C_DIS
LIN {X 0.007,Y -383.825,Z 787.622,A 0.000,B 0.000,C 90.000,E1 147.916} C_DIS
LIN {X 0.015,Y -385.857,Z 787.616,A 0.000,B 0.000,C 90.000,E1 146.834} C_DIS
LIN {X 0.041,Y -388.165,Z 787.610,A 0.000,B 0.000,C 90.000,E1 145.754} C_DIS
LIN {X -0.069,Y -390.042,Z 787.606,A 0.000,B 0.000,C 90.000,E1 145.055} C_DIS
LIN {X 0.030,Y -392.955,Z 787.601,A 0.000,B 0.000,C 90.000,E1 144.149} C_DIS
LIN {X 0.194,Y -395.894,Z 787.597,A 0.000,B 0.000,C 90.000,E1 143.417} C_DIS
LIN {X 0.049,Y -397.657,Z 787.595,A 0.000,B 0.000,C 90.000,E1 143.084} C_DIS
LIN {X -0.170,Y -399.340,Z 787.593,A 0.000,B 0.000,C 90.000,E1 142.763} C_DIS
LIN {X 0.154,Y -402.307,Z 787.590,A 0.000,B 0.000,C 90.000,E1 142.190} C_DIS
LIN {X -0.178,Y -406.358,Z 787.587,A 0.000,B 0.000,C 90.000,E1 141.618} C_DIS
LIN {X 0.056,Y -412.295,Z 787.582,A 0.000,B 0.000,C 90.000,E1 140.803} C_DIS
LIN {X 0.126,Y -427.124,Z 787.572,A 0.000,B 0.000,C 90.000,E1 139.013} C_DIS
LIN {X -0.218,Y -440.692,Z 787.564,A 0.000,B 0.000,C 90.000,E1 137.472} C_DIS
LIN {X 0.253,Y -452.471,Z 787.556,A 0.000,B 0.000,C 90.000,E1 136.053} C_DIS
LIN {X -0.120,Y -460.214,Z 787.551,A 0.000,B 0.000,C 90.000,E1 135.162} C_DIS
LIN {X -0.030,Y -466.152,Z 787.547,A 0.000,B 0.000,C 90.000,E1 134.393} C_DIS
LIN {X -0.143,Y -473.272,Z 787.541,A 0.000,B 0.000,C 90.000,E1 133.461} C_DIS
LIN {X -0.212,Y -477.920,Z 787.538,A 0.000,B 0.000,C 90.000,E1 132.852} C_DIS
LIN {X -0.090,Y -485.608,Z 787.532,A 0.000,B 0.000,C 90.000,E1 131.757} C_DIS
LIN {X -0.131,Y -489.877,Z 787.529,A 0.000,B 0.000,C 90.000,E1 131.148} C_DIS
LIN {X -0.122,Y -497.694,Z 787.522,A 0.000,B 0.000,C 90.000,E1 129.930} C_DIS
LIN {X 0.191,Y -503.220,Z 787.517,A 0.000,B 0.000,C 90.000,E1 128.991} C_DIS
LIN {X -0.028,Y -509.343,Z 787.511,A 0.000,B 0.000,C 90.000,E1 127.971} C_DIS
LIN {X -0.093,Y -513.362,Z 787.507,A 0.000,B 0.000,C 90.000,E1 127.237} C_DIS
LIN {X 0.164,Y -520.220,Z 787.500,A 0.000,B 0.000,C 90.000,E1 125.884} C_DIS
LIN {X -0.025,Y -526.077,Z 787.493,A 0.000,B 0.000,C 90.000,E1 124.739} C_DIS
LIN {X -0.068,Y -531.614,Z 787.486,A 0.000,B 0.000,C 90.000,E1 123.452} C_DIS
LIN {X 0.183,Y -535.684,Z 787.480,A 0.000,B 0.000,C 90.000,E1 122.418} C_DIS
LIN {X -0.119,Y -538.982,Z 787.475,A 0.000,B 0.000,C 90.000,E1 121.592} C_DIS
LIN {X 0.069,Y -542.119,Z 787.471,A 0.000,B 0.000,C 90.000,E1 120.718} C_DIS
LIN {X 0.018,Y -545.082,Z 787.466,A 0.000,B 0.000,C 90.000,E1 119.873} C_DIS
LIN {X 0.005,Y -547.844,Z 787.461,A 0.000,B 0.000,C 90.000,E1 119.027} C_DIS
LIN {X 0.024,Y -550.471,Z 787.457,A 0.000,B 0.000,C 90.000,E1 118.180} C_DIS
LIN {X 0.072,Y -552.936,Z 787.452,A 0.000,B 0.000,C 90.000,E1 117.334} C_DIS
LIN {X 0.142,Y -555.067,Z 787.447,A 0.000,B 0.000,C 90.000,E1 116.488} C_DIS
LIN {X -0.013,Y -556.853,Z 787.443,A 0.000,B 0.000,C 90.000,E1 115.668} C_DIS
LIN {X 0.088,Y -558.319,Z 787.438,A 0.000,B 0.000,C 90.000,E1 114.823} C_DIS
LIN {X -0.036,Y -559.497,Z 787.433,A 0.000,B 0.000,C 90.000,E1 114.003} C_DIS
LIN {X -0.270,Y -560.955,Z 787.426,A 0.000,B 0.000,C 90.000,E1 112.642} C_DIS
LIN {X 0.050,Y -562.425,Z 787.418,A 0.000,B 0.000,C 90.000,E1 111.227} C_DIS
LIN {X -0.136,Y -563.637,Z 787.410,A 0.000,B 0.000,C 90.000,E1 109.866} C_DIS
LIN {X -0.152,Y -564.633,Z 787.403,A 0.000,B 0.000,C 90.000,E1 108.489} C_DIS
LIN {X 0.190,Y -565.735,Z 787.393,A 0.000,B 0.000,C 90.000,E1 106.804} C_DIS
LIN {X 0.327,Y -567.191,Z 787.381,A 0.000,B 0.000,C 90.000,E1 104.592} C_DIS
LIN {X 0.205,Y -568.889,Z 787.369,A 0.000,B 0.000,C 90.000,E1 102.411} C_DIS
LIN {X -0.295,Y -570.447,Z 787.358,A 0.000,B 0.000,C 90.000,E1 100.546} C_DIS
LIN {X -0.196,Y -571.989,Z 787.348,A 0.000,B 0.000,C 90.000,E1 98.624} C_DIS
LIN {X -0.162,Y -572.765,Z 787.342,A 0.000,B 0.000,C 90.000,E1 97.530} C_DIS
LIN {X 0.272,Y -573.857,Z 787.333,A 0.000,B 0.000,C 90.000,E1 95.853} C_DIS
LIN {X -0.101,Y -574.615,Z 787.325,A 0.000,B 0.000,C 90.000,E1 94.531} C_DIS
LIN {X 0.076,Y -575.392,Z 787.318,A 0.000,B 0.000,C 90.000,E1 93.154} C_DIS
LIN {X 0.293,Y -576.046,Z 787.310,A 0.000,B 0.000,C 90.000,E1 91.776} C_DIS
LIN {X -0.097,Y -576.590,Z 787.303,A 0.000,B 0.000,C 90.000,E1 90.458} C_DIS
LIN {X 0.259,Y -577.277,Z 787.294,A 0.000,B 0.000,C 90.000,E1 88.797} C_DIS
LIN {X -0.095,Y -577.661,Z 787.286,A 0.000,B 0.000,C 90.000,E1 87.478} C_DIS
LIN {X 0.134,Y -578.029,Z 787.278,A 0.000,B 0.000,C 90.000,E1 86.102} C_DIS
LIN {X 0.032,Y -578.342,Z 787.269,A 0.000,B 0.000,C 90.000,E1 84.489} C_DIS
LIN {X -0.054,Y -578.652,Z 787.260,A 0.000,B 0.000,C 90.000,E1 82.875} C_DIS
LIN {X -0.281,Y -578.867,Z 787.253,A 0.000,B 0.000,C 90.000,E1 81.546} C_DIS
LIN {X -0.067,Y -579.000,Z 787.247,A 0.000,B 0.000,C 90.000,E1 80.443} C_DIS
LIN {X -0.202,Y -579.144,Z 787.239,A 0.000,B 0.000,C 90.000,E1 79.106} C_DIS
LIN {X 0.119,Y -579.149,Z 787.233,A 0.000,B 0.000,C 90.000,E1 77.993} C_DIS
LIN {X 0.096,Y -579.046,Z 787.226,A 0.000,B 0.000,C 90.000,E1 76.645} C_DIS
LIN {X 0.206,Y -578.834,Z 787.218,A 0.000,B 0.000,C 90.000,E1 75.283} C_DIS
LIN {X 0.334,Y -578.399,Z 787.208,A 0.000,B 0.000,C 90.000,E1 73.378} C_DIS
LIN {X 0.213,Y -578.093,Z 787.202,A 0.000,B 0.000,C 90.000,E1 72.308} C_DIS
LIN {X 0.067,Y -577.871,Z 787.197,A 0.000,B 0.000,C 90.000,E1 71.511} C_DIS
LIN {X -0.028,Y -577.050,Z 787.187,A 0.000,B 0.000,C 90.000,E1 69.625} C_DIS
LIN {X 0.213,Y -576.188,Z 787.178,A 0.000,B 0.000,C 90.000,E1 67.975} C_DIS
LIN {X 0.268,Y -575.380,Z 787.170,A 0.000,B 0.000,C 90.000,E1 66.613} C_DIS
LIN {X 0.014,Y -574.369,Z 787.163,A 0.000,B 0.000,C 90.000,E1 65.281} C_DIS
LIN {X -0.092,Y -573.542,Z 787.157,A 0.000,B 0.000,C 90.000,E1 64.204} C_DIS
LIN {X 0.134,Y -572.180,Z 787.149,A 0.000,B 0.000,C 90.000,E1 62.820} C_DIS
LIN {X -0.260,Y -570.873,Z 787.143,A 0.000,B 0.000,C 90.000,E1 61.769} C_DIS
LIN {X -0.060,Y -568.939,Z 787.135,A 0.000,B 0.000,C 90.000,E1 60.383} C_DIS
LIN {X 0.183,Y -567.631,Z 787.131,A 0.000,B 0.000,C 90.000,E1 59.537} C_DIS
LIN {X 0.021,Y -565.593,Z 787.125,A 0.000,B 0.000,C 90.000,E1 58.456} C_DIS
LIN {X -0.265,Y -563.925,Z 787.120,A 0.000,B 0.000,C 90.000,E1 57.661} C_DIS
LIN {X -0.268,Y -562.039,Z 787.116,A 0.000,B 0.000,C 90.000,E1 56.834} C_DIS
LIN {X 0.175,Y -559.940,Z 787.111,A 0.000,B 0.000,C 90.000,E1 55.960} C_DIS
LIN {X -0.333,Y -557.635,Z 787.106,A 0.000,B 0.000,C 90.000,E1 55.182} C_DIS
LIN {X -0.003,Y -554.160,Z 787.100,A 0.000,B 0.000,C 90.000,E1 54.036} C_DIS
LIN {X -0.183,Y -552.295,Z 787.097,A 0.000,B 0.000,C 90.000,E1 53.497} C_DIS
LIN {X -0.051,Y -550.298,Z 787.094,A 0.000,B 0.000,C 90.000,E1 52.924} C_DIS
LIN {X 0.116,Y -546.898,Z 787.089,A 0.000,B 0.000,C 90.000,E1 52.065} C_DIS
LIN {X -0.032,Y -543.835,Z 787.085,A 0.000,B 0.000,C 90.000,E1 51.376} C_DIS
LIN {X 0.217,Y -540.506,Z 787.082,A 0.000,B 0.000,C 90.000,E1 50.642} C_DIS
LIN {X -0.161,Y -537.590,Z 787.078,A 0.000,B 0.000,C 90.000,E1 50.114} C_DIS
LIN {X -0.146,Y -534.414,Z 787.075,A 0.000,B 0.000,C 90.000,E1 49.542} C_DIS
LIN {X 0.187,Y -530.918,Z 787.072,A 0.000,B 0.000,C 90.000,E1 48.933} C_DIS
LIN {X -0.255,Y -527.009,Z 787.069,A 0.000,B 0.000,C 90.000,E1 48.405} C_DIS
LIN {X 0.020,Y -522.636,Z 787.066,A 0.000,B 0.000,C 90.000,E1 47.796} C_DIS
LIN {X 0.022,Y -517.962,Z 787.062,A 0.000,B 0.000,C 90.000,E1 47.229} C_DIS
LIN {X 0.054,Y -512.932,Z 787.059,A 0.000,B 0.000,C 90.000,E1 46.662} C_DIS
LIN {X 0.220,Y -508.880,Z 787.057,A 0.000,B 0.000,C 90.000,E1 46.215} C_DIS
LIN {X -0.297,Y -503.187,Z 787.054,A 0.000,B 0.000,C 90.000,E1 45.729} C_DIS
LIN {X -0.211,Y -498.741,Z 787.052,A 0.000,B 0.000,C 90.000,E1 45.324} C_DIS
LIN {X -0.222,Y -493.012,Z 787.049,A 0.000,B 0.000,C 90.000,E1 44.838} C_DIS
LIN {X 0.127,Y -485.186,Z 787.046,A 0.000,B 0.000,C 90.000,E1 44.190} C_DIS
LIN {X 0.256,Y -477.693,Z 787.043,A 0.000,B 0.000,C 90.000,E1 43.623} C_DIS
LIN {X -0.090,Y -464.761,Z 787.038,A 0.000,B 0.000,C 90.000,E1 42.771} C_DIS
LIN {X -0.251,Y -451.814,Z 787.033,A 0.000,B 0.000,C 90.000,E1 41.919} C_DIS
LIN {X -0.041,Y -421.782,Z 787.021,A 0.000,B 0.000,C 90.000,E1 39.725} C_DIS
LIN {X 0.007,Y -410.961,Z 787.016,A 0.000,B 0.000,C 90.000,E1 38.830} C_DIS
LIN {X -0.073,Y -405.448,Z 787.013,A 0.000,B 0.000,C 90.000,E1 38.302} C_DIS
LIN {X -0.106,Y -405.422,Z 787.013,A 0.000,B 0.000,C 90.000,E1 38.302} C_DIS
LIN {X 0.026,Y -396.784,Z 786.988,A 0.000,B 0.000,C 90.000,E1 33.833} C_DIS
LIN {X -0.100,Y -396.219,Z 786.986,A 0.000,B 0.000,C 90.000,E1 33.499} C_DIS
LIN {X -0.026,Y -396.968,Z 786.970,A 0.000,B 0.000,C 90.000,E1 30.669} C_DIS
LIN {X 0.020,Y -398.299,Z 786.955,A 0.000,B 0.000,C 90.000,E1 27.847} C_DIS
LIN {X -0.143,Y -399.702,Z 786.941,A 0.000,B 0.000,C 90.000,E1 25.412} C_DIS
LIN {X -0.081,Y -401.367,Z 786.927,A 0.000,B 0.000,C 90.000,E1 22.950} C_DIS
LIN {X -0.107,Y -404.084,Z 786.910,A 0.000,B 0.000,C 90.000,E1 19.812} C_DIS
LIN {X 0.177,Y -409.079,Z 786.887,A 0.000,B 0.000,C 90.000,E1 15.607} C_DIS
LIN {X -0.019,Y -413.787,Z 786.870,A 0.000,B 0.000,C 90.000,E1 12.535} C_DIS
LIN {X -0.071,Y -417.300,Z 786.858,A 0.000,B 0.000,C 90.000,E1 10.489} C_DIS
LIN {X -0.115,Y -420.845,Z 786.847,A 0.000,B 0.000,C 90.000,E1 8.454} C_DIS
LIN {X 0.198,Y -423.845,Z 786.838,A 0.000,B 0.000,C 90.000,E1 6.720} C_DIS
LIN {X -0.185,Y -428.080,Z 786.824,A 0.000,B 0.000,C 90.000,E1 4.416} C_DIS
LIN {X -0.087,Y -432.482,Z 786.811,A 0.000,B 0.000,C 90.000,E1 2.064} C_DIS
LIN {X 0.165,Y -437.030,Z 786.799,A 0.000,B 0.000,C 90.000,E1 359.771} C_DIS
LIN {X 0.185,Y -442.719,Z 786.784,A 0.000,B 0.000,C 90.000,E1 357.135} C_DIS
LIN {X -0.161,Y -448.074,Z 786.772,A 0.000,B 0.000,C 90.000,E1 354.894} C_DIS
LIN {X 0.125,Y -453.475,Z 786.759,A 0.000,B 0.000,C 90.000,E1 352.591} C_DIS
LIN {X -0.227,Y -457.259,Z 786.750,A 0.000,B 0.000,C 90.000,E1 351.027} C_DIS
LIN {X 0.051,Y -462.557,Z 786.738,A 0.000,B 0.000,C 90.000,E1 348.757} C_DIS
LIN {X 0.090,Y -464.240,Z 786.734,A 0.000,B 0.000,C 90.000,E1 348.117} C_DIS
LIN {X -0.015,Y -465.211,Z 786.732,A 0.000,B 0.000,C 90.000,E1 347.813} C_DIS
LIN {X -0.135,Y -466.978,Z 786.730,A 0.000,B 0.000,C 90.000,E1 347.353} C_DIS
LIN {X -0.015,Y -468.881,Z 786.727,A 0.000,B 0.000,C 90.000,E1 346.937} C_DIS
LIN {X -0.012,Y -471.987,Z 786.725,A 0.000,B 0.000,C 90.000,E1 346.464} C_DIS
LIN {X 0.072,Y -476.386,Z 786.722,A 0.000,B 0.000,C 90.000,E1 345.936} C_DIS
LIN {X -0.227,Y -482.421,Z 786.719,A 0.000,B 0.000,C 90.000,E1 345.408} C_DIS
LIN {X 0.097,Y -494.419,Z 786.714,A 0.000,B 0.000,C 90.000,E1 344.464} C_DIS
LIN {X -0.264,Y -514.929,Z 786.706,A 0.000,B 0.000,C 90.000,E1 343.087} C_DIS
LIN {X 0.182,Y -530.759,Z 786.700,A 0.000,B 0.000,C 90.000,E1 342.000} C_DIS
LIN {X -0.100,Y -538.516,Z 786.697,A 0.000,B 0.000,C 90.000,E1 341.511} C_DIS
LIN {X 0.002,Y -547.633,Z 786.694,A 0.000,B 0.000,C 90.000,E1 340.859} C_DIS
LIN {X 0.011,Y -554.957,Z 786.691,A 0.000,B 0.000,C 90.000,E1 340.296} C_DIS
LIN {X -0.050,Y -560.432,Z 786.688,A 0.000,B 0.000,C 90.000,E1 339.826} C_DIS
LIN {X -0.217,Y -566.925,Z 786.684,A 0.000,B 0.000,C 90.000,E1 339.209} C_DIS
LIN {X 0.074,Y -571.856,Z 786.681,A 0.000,B 0.000,C 90.000,E1 338.646} C_DIS
LIN {X -0.026,Y -577.528,Z 786.678,A 0.000,B 0.000,C 90.000,E1 337.975} C_DIS
LIN {X -0.090,Y -582.890,Z 786.674,A 0.000,B 0.000,C 90.000,E1 337.305} C_DIS
LIN {X 0.053,Y -588.846,Z 786.669,A 0.000,B 0.000,C 90.000,E1 336.485} C_DIS
LIN {X 0.174,Y -596.220,Z 786.664,A 0.000,B 0.000,C 90.000,E1 335.409} C_DIS
LIN {X -0.367,Y -602.371,Z 786.658,A 0.000,B 0.000,C 90.000,E1 334.537} C_DIS
LIN {X -0.067,Y -608.977,Z 786.653,A 0.000,B 0.000,C 90.000,E1 333.461} C_DIS
LIN {X 0.075,Y -614.429,Z 786.648,A 0.000,B 0.000,C 90.000,E1 332.538} C_DIS
LIN {X 0.001,Y -619.618,Z 786.643,A 0.000,B 0.000,C 90.000,E1 331.641} C_DIS
LIN {X 0.286,Y -625.311,Z 786.637,A 0.000,B 0.000,C 90.000,E1 330.589} C_DIS
LIN {X 0.108,Y -630.689,Z 786.631,A 0.000,B 0.000,C 90.000,E1 329.587} C_DIS
LIN {X -0.345,Y -635.216,Z 786.626,A 0.000,B 0.000,C 90.000,E1 328.742} C_DIS
LIN {X -0.087,Y -639.396,Z 786.621,A 0.000,B 0.000,C 90.000,E1 327.837} C_DIS
LIN {X -0.094,Y -643.913,Z 786.616,A 0.000,B 0.000,C 90.000,E1 326.834} C_DIS
LIN {X -0.170,Y -646.034,Z 786.613,A 0.000,B 0.000,C 90.000,E1 326.342} C_DIS
LIN {X 0.264,Y -650.134,Z 786.607,A 0.000,B 0.000,C 90.000,E1 325.308} C_DIS
LIN {X -0.164,Y -653.935,Z 786.602,A 0.000,B 0.000,C 90.000,E1 324.356} C_DIS
LIN {X 0.219,Y -657.497,Z 786.596,A 0.000,B 0.000,C 90.000,E1 323.336} C_DIS
LIN {X 0.218,Y -661.604,Z 786.590,A 0.000,B 0.000,C 90.000,E1 322.110} C_DIS
LIN {X -0.216,Y -664.659,Z 786.584,A 0.000,B 0.000,C 90.000,E1 321.170} C_DIS
LIN {X -0.195,Y -667.529,Z 786.579,A 0.000,B 0.000,C 90.000,E1 320.194} C_DIS
LIN {X -0.132,Y -670.256,Z 786.573,A 0.000,B 0.000,C 90.000,E1 319.218} C_DIS
LIN {X -0.050,Y -672.164,Z 786.569,A 0.000,B 0.000,C 90.000,E1 318.485} C_DIS
LIN {X 0.016,Y -674.671,Z 786.564,A 0.000,B 0.000,C 90.000,E1 317.514} C_DIS
LIN {X 0.189,Y -677.297,Z 786.557,A 0.000,B 0.000,C 90.000,E1 316.296} C_DIS
LIN {X -0.024,Y -680.443,Z 786.548,A 0.000,B 0.000,C 90.000,E1 314.636} C_DIS
LIN {X -0.364,Y -681.652,Z 786.544,A 0.000,B 0.000,C 90.000,E1 313.947} C_DIS
LIN {X -0.025,Y -683.952,Z 786.536,A 0.000,B 0.000,C 90.000,E1 312.486} C_DIS
LIN {X -0.204,Y -685.637,Z 786.529,A 0.000,B 0.000,C 90.000,E1 311.310} C_DIS
LIN {X 0.149,Y -687.121,Z 786.523,A 0.000,B 0.000,C 90.000,E1 310.092} C_DIS
LIN {X 0.085,Y -688.425,Z 786.516,A 0.000,B 0.000,C 90.000,E1 308.910} C_DIS
LIN {X -0.099,Y -690.316,Z 786.506,A 0.000,B 0.000,C 90.000,E1 307.030} C_DIS
LIN {X 0.068,Y -691.557,Z 786.498,A 0.000,B 0.000,C 90.000,E1 305.598} C_DIS
LIN {X -0.150,Y -692.642,Z 786.490,A 0.000,B 0.000,C 90.000,E1 304.199} C_DIS
LIN {X -0.129,Y -693.849,Z 786.481,A 0.000,B 0.000,C 90.000,E1 302.546} C_DIS
LIN {X -0.108,Y -694.984,Z 786.473,A 0.000,B 0.000,C 90.000,E1 301.131} C_DIS
LIN {X -0.318,Y -695.649,Z 786.468,A 0.000,B 0.000,C 90.000,E1 300.207} C_DIS
LIN {X 0.328,Y -696.375,Z 786.460,A 0.000,B 0.000,C 90.000,E1 298.743} C_DIS
LIN {X 0.060,Y -696.974,Z 786.453,A 0.000,B 0.000,C 90.000,E1 297.590} C_DIS
LIN {X 0.238,Y -698.226,Z 786.442,A 0.000,B 0.000,C 90.000,E1 295.463} C_DIS
LIN {X 0.102,Y -698.692,Z 786.438,A 0.000,B 0.000,C 90.000,E1 294.771} C_DIS
LIN {X -0.295,Y -698.746,Z 786.435,A 0.000,B 0.000,C 90.000,E1 294.335} C_DIS
LIN {X -0.031,Y -698.598,Z 786.434,A 0.000,B 0.000,C 90.000,E1 294.079} C_DIS
LIN {X 0.215,Y -697.666,Z 786.431,A 0.000,B 0.000,C 90.000,E1 293.590} C_DIS
LIN {X -0.165,Y -696.848,Z 786.430,A 0.000,B 0.000,C 90.000,E1 293.387} C_DIS
LIN {X 0.070,Y -693.343,Z 786.427,A 0.000,B 0.000,C 90.000,E1 292.898} C_DIS
LIN {X 0.192,Y -692.332,Z 786.427,A 0.000,B 0.000,C 90.000,E1 292.770} C_DIS
LIN {X 0.313,Y -690.956,Z 786.426,A 0.000,B 0.000,C 90.000,E1 292.642} C_DIS
LIN {X -0.372,Y -688.915,Z 786.425,A 0.000,B 0.000,C 90.000,E1 292.589} C_DIS
LIN {X -0.349,Y -683.183,Z 786.424,A 0.000,B 0.000,C 90.000,E1 292.333} C_DIS
LIN {X 0.321,Y -681.186,Z 786.424,A 0.000,B 0.000,C 90.000,E1 292.206} C_DIS
LIN {X -0.143,Y -674.937,Z 786.423,A 0.000,B 0.000,C 90.000,E1 292.078} C_DIS
LIN {X -0.066,Y -672.832,Z 786.422,A 0.000,B 0.000,C 90.000,E1 292.025} C_DIS
LIN {X -0.239,Y -655.840,Z 786.421,A 0.000,B 0.000,C 90.000,E1 291.770} C_DIS
LIN {X 0.195,Y -638.258,Z 786.419,A 0.000,B 0.000,C 90.000,E1 291.408} C_DIS
LIN {X -0.003,Y -617.492,Z 786.417,A 0.000,B 0.000,C 90.000,E1 290.972} C_DIS
LIN {X -0.142,Y -600.223,Z 786.414,A 0.000,B 0.000,C 90.000,E1 290.556} C_DIS
LIN {X -0.075,Y -583.456,Z 786.411,A 0.000,B 0.000,C 90.000,E1 290.066} C_DIS
LIN {X -0.185,Y -569.871,Z 786.409,A 0.000,B 0.000,C 90.000,E1 289.631} C_DIS
LIN {X -0.172,Y -565.325,Z 786.408,A 0.000,B 0.000,C 90.000,E1 289.450} C_DIS
LIN {X 0.164,Y -562.334,Z 786.407,A 0.000,B 0.000,C 90.000,E1 289.268} C_DIS
LIN {X 0.247,Y -558.334,Z 786.406,A 0.000,B 0.000,C 90.000,E1 288.960} C_DIS
LIN {X -0.294,Y -556.590,Z 786.404,A 0.000,B 0.000,C 90.000,E1 288.725} C_DIS
LIN {X -0.122,Y -555.262,Z 786.402,A 0.000,B 0.000,C 90.000,E1 288.290} C_DIS
LIN {X -0.134,Y -554.660,Z 786.399,A 0.000,B 0.000,C 90.000,E1 287.873} C_DIS
LIN {X 0.110,Y -552.849,Z 786.378,A 0.000,B 0.000,C 90.000,E1 283.939} C_DIS
LIN {X -0.254,Y -552.323,Z 786.368,A 0.000,B 0.000,C 90.000,E1 282.299} C_DIS
LIN {X 0.037,Y -551.741,Z 786.357,A 0.000,B 0.000,C 90.000,E1 280.310} C_DIS
LIN {X -0.023,Y -551.307,Z 786.350,A 0.000,B 0.000,C 90.000,E1 278.916} C_DIS
LIN {X -0.059,Y -550.941,Z 786.340,A 0.000,B 0.000,C 90.000,E1 277.239} C_DIS
LIN {X 0.234,Y -550.433,Z 786.334,A 0.000,B 0.000,C 90.000,E1 276.087} C_DIS
LIN {X 0.066,Y -549.686,Z 786.326,A 0.000,B 0.000,C 90.000,E1 274.702} C_DIS
LIN {X -0.206,Y -548.729,Z 786.318,A 0.000,B 0.000,C 90.000,E1 273.326} C_DIS
LIN {X 0.176,Y -547.507,Z 786.307,A 0.000,B 0.000,C 90.000,E1 271.318} C_DIS
LIN {X -0.098,Y -546.428,Z 786.298,A 0.000,B 0.000,C 90.000,E1 269.656} C_DIS
LIN {X 0.164,Y -545.233,Z 786.289,A 0.000,B 0.000,C 90.000,E1 267.936} C_DIS
LIN {X -0.117,Y -543.948,Z 786.278,A 0.000,B 0.000,C 90.000,E1 265.988} C_DIS
LIN {X 0.045,Y -543.459,Z 786.273,A 0.000,B 0.000,C 90.000,E1 265.122} C_DIS
LIN {X 0.245,Y -542.536,Z 786.265,A 0.000,B 0.000,C 90.000,E1 263.685} C_DIS
LIN {X -0.057,Y -541.398,Z 786.257,A 0.000,B 0.000,C 90.000,E1 262.299} C_DIS
LIN {X -0.241,Y -539.742,Z 786.246,A 0.000,B 0.000,C 90.000,E1 260.330} C_DIS
LIN {X 0.043,Y -538.726,Z 786.240,A 0.000,B 0.000,C 90.000,E1 259.162} C_DIS
LIN {X -0.080,Y -537.094,Z 786.230,A 0.000,B 0.000,C 90.000,E1 257.465} C_DIS
LIN {X -0.177,Y -535.729,Z 786.222,A 0.000,B 0.000,C 90.000,E1 256.047} C_DIS
LIN {X -0.064,Y -533.530,Z 786.211,A 0.000,B 0.000,C 90.000,E1 254.031} C_DIS
LIN {X -0.058,Y -531.578,Z 786.202,A 0.000,B 0.000,C 90.000,E1 252.308} C_DIS
LIN {X 0.035,Y -529.847,Z 786.194,A 0.000,B 0.000,C 90.000,E1 250.859} C_DIS
LIN {X 0.272,Y -527.822,Z 786.186,A 0.000,B 0.000,C 90.000,E1 249.390} C_DIS
LIN {X 0.155,Y -525.332,Z 786.176,A 0.000,B 0.000,C 90.000,E1 247.667} C_DIS
LIN {X -0.141,Y -523.533,Z 786.170,A 0.000,B 0.000,C 90.000,E1 246.538} C_DIS
LIN {X 0.018,Y -521.788,Z 786.163,A 0.000,B 0.000,C 90.000,E1 245.357} C_DIS
LIN {X 0.036,Y -519.418,Z 786.155,A 0.000,B 0.000,C 90.000,E1 243.896} C_DIS
LIN {X -0.121,Y -517.484,Z 786.149,A 0.000,B 0.000,C 90.000,E1 242.743} C_DIS
LIN {X 0.028,Y -515.952,Z 786.144,A 0.000,B 0.000,C 90.000,E1 241.847} C_DIS
LIN {X -0.036,Y -513.179,Z 786.135,A 0.000,B 0.000,C 90.000,E1 240.383} C_DIS
LIN {X -0.139,Y -510.443,Z 786.127,A 0.000,B 0.000,C 90.000,E1 238.918} C_DIS
LIN {X 0.026,Y -506.804,Z 786.117,A 0.000,B 0.000,C 90.000,E1 237.120} C_DIS
LIN {X 0.030,Y -504.255,Z 786.111,A 0.000,B 0.000,C 90.000,E1 235.928} C_DIS
LIN {X -0.285,Y -501.525,Z 786.104,A 0.000,B 0.000,C 90.000,E1 234.769} C_DIS
LIN {X 0.060,Y -499.357,Z 786.099,A 0.000,B 0.000,C 90.000,E1 233.829} C_DIS
LIN {X -0.179,Y -495.591,Z 786.091,A 0.000,B 0.000,C 90.000,E1 232.351} C_DIS
LIN {X 0.120,Y -490.331,Z 786.079,A 0.000,B 0.000,C 90.000,E1 230.194} C_DIS
LIN {X -0.128,Y -484.068,Z 786.064,A 0.000,B 0.000,C 90.000,E1 227.472} C_DIS
LIN {X 0.218,Y -480.774,Z 786.055,A 0.000,B 0.000,C 90.000,E1 225.891} C_DIS
LIN {X 0.271,Y -476.651,Z 786.045,A 0.000,B 0.000,C 90.000,E1 224.028} C_DIS
LIN {X -0.198,Y -473.276,Z 786.036,A 0.000,B 0.000,C 90.000,E1 222.528} C_DIS
LIN {X -0.106,Y -467.903,Z 786.022,A 0.000,B 0.000,C 90.000,E1 220.011} C_DIS
LIN {X 0.028,Y -464.607,Z 786.013,A 0.000,B 0.000,C 90.000,E1 218.418} C_DIS
LIN {X 0.131,Y -460.636,Z 786.003,A 0.000,B 0.000,C 90.000,E1 216.503} C_DIS
LIN {X 0.062,Y -455.977,Z 785.991,A 0.000,B 0.000,C 90.000,E1 214.278} C_DIS
LIN {X 0.062,Y -452.725,Z 785.982,A 0.000,B 0.000,C 90.000,E1 212.673} C_DIS
LIN {X -0.021,Y -448.951,Z 785.971,A 0.000,B 0.000,C 90.000,E1 210.747} C_DIS
LIN {X -0.183,Y -445.195,Z 785.960,A 0.000,B 0.000,C 90.000,E1 208.821} C_DIS
LIN {X -0.108,Y -442.105,Z 785.951,A 0.000,B 0.000,C 90.000,E1 207.180} C_DIS
LIN {X -0.102,Y -438.968,Z 785.942,A 0.000,B 0.000,C 90.000,E1 205.540} C_DIS
LIN {X -0.141,Y -435.269,Z 785.931,A 0.000,B 0.000,C 90.000,E1 203.567} C_DIS
LIN {X -0.004,Y -430.767,Z 785.918,A 0.000,B 0.000,C 90.000,E1 201.227} C_DIS
LIN {X -0.161,Y -428.882,Z 785.912,A 0.000,B 0.000,C 90.000,E1 200.248} C_DIS
LIN {X 0.050,Y -424.415,Z 785.899,A 0.000,B 0.000,C 90.000,E1 197.873} C_DIS
LIN {X 0.097,Y -420.474,Z 785.888,A 0.000,B 0.000,C 90.000,E1 195.843} C_DIS
LIN {X 0.181,Y -414.672,Z 785.871,A 0.000,B 0.000,C 90.000,E1 192.771} C_DIS
LIN {X -0.005,Y -412.779,Z 785.865,A 0.000,B 0.000,C 90.000,E1 191.771} C_DIS
LIN {X -0.106,Y -406.682,Z 785.846,A 0.000,B 0.000,C 90.000,E1 188.341} C_DIS
LIN {X -0.060,Y -404.335,Z 785.839,A 0.000,B 0.000,C 90.000,E1 186.947} C_DIS
LIN {X -0.206,Y -400.739,Z 785.827,A 0.000,B 0.000,C 90.000,E1 184.878} C_DIS
LIN {X -0.060,Y -394.137,Z 785.802,A 0.000,B 0.000,C 90.000,E1 180.286} C_DIS
LIN {X -0.088,Y -391.719,Z 785.790,A 0.000,B 0.000,C 90.000,E1 178.165} C_DIS
LIN {X -0.088,Y -389.969,Z 785.780,A 0.000,B 0.000,C 90.000,E1 176.388} C_DIS
LIN {X -0.110,Y -388.208,Z 785.770,A 0.000,B 0.000,C 90.000,E1 174.609} C_DIS
LIN {X -0.041,Y -385.108,Z 785.752,A 0.000,B 0.000,C 90.000,E1 171.376} C_DIS
LIN {X 0.173,Y -382.755,Z 785.736,A 0.000,B 0.000,C 90.000,E1 168.465} C_DIS
LIN {X 0.090,Y -380.929,Z 785.720,A 0.000,B 0.000,C 90.000,E1 165.589} C_DIS
LIN {X -0.129,Y -379.474,Z 785.704,A 0.000,B 0.000,C 90.000,E1 162.725} C_DIS
LIN {X -0.163,Y -378.543,Z 785.688,A 0.000,B 0.000,C 90.000,E1 159.826} C_DIS
LIN {X 0.178,Y -378.195,Z 785.674,A 0.000,B 0.000,C 90.000,E1 157.230} C_DIS
LIN {X 0.026,Y -379.081,Z 785.651,A 0.000,B 0.000,C 90.000,E1 153.256} C_DIS
LIN {X 0.163,Y -380.887,Z 785.635,A 0.000,B 0.000,C 90.000,E1 150.333} C_DIS
LIN {X -0.050,Y -382.498,Z 785.627,A 0.000,B 0.000,C 90.000,E1 148.918} C_DIS
LIN {X 0.092,Y -384.562,Z 785.619,A 0.000,B 0.000,C 90.000,E1 147.454} C_DIS
LIN {X 0.037,Y -388.920,Z 785.607,A 0.000,B 0.000,C 90.000,E1 145.308} C_DIS
LIN {X -0.065,Y -390.938,Z 785.603,A 0.000,B 0.000,C 90.000,E1 144.609} C_DIS
LIN {X -0.029,Y -392.709,Z 785.600,A 0.000,B 0.000,C 90.000,E1 144.069} C_DIS
LIN {X -0.071,Y -394.760,Z 785.597,A 0.000,B 0.000,C 90.000,E1 143.543} C_DIS
LIN {X -0.124,Y -397.919,Z 785.594,A 0.000,B 0.000,C 90.000,E1 142.844} C_DIS
LIN {X 0.088,Y -401.772,Z 785.590,A 0.000,B 0.000,C 90.000,E1 142.110} C_DIS
LIN {X -0.236,Y -405.713,Z 785.586,A 0.000,B 0.000,C 90.000,E1 141.537} C_DIS
LIN {X -0.057,Y -410.402,Z 785.583,A 0.000,B 0.000,C 90.000,E1 140.884} C_DIS
LIN {X -0.010,Y -423.853,Z 785.574,A 0.000,B 0.000,C 90.000,E1 139.256} C_DIS
LIN {X -0.184,Y -432.043,Z 785.568,A 0.000,B 0.000,C 90.000,E1 138.324} C_DIS
LIN {X -0.014,Y -440.042,Z 785.563,A 0.000,B 0.000,C 90.000,E1 137.391} C_DIS
LIN {X 0.200,Y -450.888,Z 785.557,A 0.000,B 0.000,C 90.000,E1 136.134} C_DIS
LIN {X -0.225,Y -456.133,Z 785.553,A 0.000,B 0.000,C 90.000,E1 135.567} C_DIS
LIN {X -0.132,Y -461.368,Z 785.549,A 0.000,B 0.000,C 90.000,E1 134.919} C_DIS
LIN {X -0.034,Y -466.369,Z 785.546,A 0.000,B 0.000,C 90.000,E1 134.271} C_DIS
LIN {X 0.003,Y -477.113,Z 785.538,A 0.000,B 0.000,C 90.000,E1 132.852} C_DIS
LIN {X -0.042,Y -482.736,Z 785.534,A 0.000,B 0.000,C 90.000,E1 132.081} C_DIS
LIN {X 0.117,Y -490.288,Z 785.528,A 0.000,B 0.000,C 90.000,E1 130.987} C_DIS
LIN {X -0.184,Y -498.162,Z 785.521,A 0.000,B 0.000,C 90.000,E1 129.806} C_DIS
LIN {X -0.036,Y -502.777,Z 785.517,A 0.000,B 0.000,C 90.000,E1 129.036} C_DIS
LIN {X 0.133,Y -508.969,Z 785.511,A 0.000,B 0.000,C 90.000,E1 127.971} C_DIS
LIN {X 0.064,Y -513.032,Z 785.507,A 0.000,B 0.000,C 90.000,E1 127.237} C_DIS
LIN {X -0.100,Y -519.944,Z 785.500,A 0.000,B 0.000,C 90.000,E1 125.931} C_DIS
LIN {X -0.002,Y -525.079,Z 785.494,A 0.000,B 0.000,C 90.000,E1 124.898} C_DIS
LIN {X -0.207,Y -527.067,Z 785.492,A 0.000,B 0.000,C 90.000,E1 124.485} C_DIS
LIN {X -0.009,Y -531.452,Z 785.486,A 0.000,B 0.000,C 90.000,E1 123.452} C_DIS
LIN {X -0.058,Y -534.974,Z 785.481,A 0.000,B 0.000,C 90.000,E1 122.594} C_DIS
LIN {X 0.082,Y -538.350,Z 785.476,A 0.000,B 0.000,C 90.000,E1 121.720} C_DIS
LIN {X -0.009,Y -542.536,Z 785.470,A 0.000,B 0.000,C 90.000,E1 120.590} C_DIS
LIN {X -0.040,Y -546.410,Z 785.464,A 0.000,B 0.000,C 90.000,E1 119.461} C_DIS
LIN {X -0.286,Y -549.981,Z 785.457,A 0.000,B 0.000,C 90.000,E1 118.359} C_DIS
LIN {X 0.013,Y -553.272,Z 785.451,A 0.000,B 0.000,C 90.000,E1 117.206} C_DIS
LIN {X 0.086,Y -555.358,Z 785.447,A 0.000,B 0.000,C 90.000,E1 116.360} C_DIS
LIN {X -0.066,Y -557.089,Z 785.442,A 0.000,B 0.000,C 90.000,E1 115.540} C_DIS
LIN {X 0.037,Y -558.510,Z 785.437,A 0.000,B 0.000,C 90.000,E1 114.695} C_DIS
LIN {X -0.314,Y -559.640,Z 785.433,A 0.000,B 0.000,C 90.000,E1 113.898} C_DIS
LIN {X 0.199,Y -561.126,Z 785.425,A 0.000,B 0.000,C 90.000,E1 112.461} C_DIS
LIN {X 0.208,Y -562.330,Z 785.419,A 0.000,B 0.000,C 90.000,E1 111.354} C_DIS
LIN {X 0.025,Y -563.593,Z 785.411,A 0.000,B 0.000,C 90.000,E1 109.993} C_DIS
LIN {X 0.192,Y -564.657,Z 785.404,A 0.000,B 0.000,C 90.000,E1 108.598} C_DIS
LIN {X -0.180,Y -565.829,Z 785.394,A 0.000,B 0.000,C 90.000,E1 106.985} C_DIS
LIN {X -0.207,Y -567.120,Z 785.384,A 0.000,B 0.000,C 90.000,E1 105.064} C_DIS
LIN {X 0.223,Y -568.780,Z 785.371,A 0.000,B 0.000,C 90.000,E1 102.827} C_DIS
LIN {X 0.210,Y -570.121,Z 785.362,A 0.000,B 0.000,C 90.000,E1 101.186} C_DIS
LIN {X 0.210,Y -570.820,Z 785.358,A 0.000,B 0.000,C 90.000,E1 100.366} C_DIS
LIN {X 0.227,Y -572.389,Z 785.347,A 0.000,B 0.000,C 90.000,E1 98.454} C_DIS
LIN {X -0.104,Y -573.357,Z 785.340,A 0.000,B 0.000,C 90.000,E1 97.125} C_DIS
LIN {X 0.150,Y -574.266,Z 785.332,A 0.000,B 0.000,C 90.000,E1 95.739} C_DIS
LIN {X -0.073,Y -575.179,Z 785.323,A 0.000,B 0.000,C 90.000,E1 94.131} C_DIS
LIN {X 0.151,Y -575.931,Z 785.315,A 0.000,B 0.000,C 90.000,E1 92.751} C_DIS
LIN {X -0.226,Y -576.592,Z 785.308,A 0.000,B 0.000,C 90.000,E1 91.432} C_DIS
LIN {X 0.285,Y -577.379,Z 785.297,A 0.000,B 0.000,C 90.000,E1 89.484} C_DIS
LIN {X -0.066,Y -577.844,Z 785.290,A 0.000,B 0.000,C 90.000,E1 88.165} C_DIS
LIN {X 0.176,Y -578.235,Z 785.282,A 0.000,B 0.000,C 90.000,E1 86.788} C_DIS
LIN {X 0.039,Y -578.624,Z 785.273,A 0.000,B 0.000,C 90.000,E1 85.179} C_DIS
LIN {X -0.103,Y -578.884,Z 785.264,A 0.000,B 0.000,C 90.000,E1 83.571} C_DIS
LIN {X 0.243,Y -579.164,Z 785.257,A 0.000,B 0.000,C 90.000,E1 82.186} C_DIS
LIN {X 0.232,Y -579.333,Z 785.248,A 0.000,B 0.000,C 90.000,E1 80.566} C_DIS
LIN {X 0.202,Y -579.476,Z 785.240,A 0.000,B 0.000,C 90.000,E1 79.218} C_DIS
LIN {X 0.069,Y -579.482,Z 785.233,A 0.000,B 0.000,C 90.000,E1 77.881} C_DIS
LIN {X 0.046,Y -579.326,Z 785.225,A 0.000,B 0.000,C 90.000,E1 76.533} C_DIS
LIN {X 0.153,Y -579.094,Z 785.218,A 0.000,B 0.000,C 90.000,E1 75.172} C_DIS
LIN {X -0.276,Y -578.636,Z 785.207,A 0.000,B 0.000,C 90.000,E1 73.323} C_DIS
LIN {X -0.220,Y -578.302,Z 785.201,A 0.000,B 0.000,C 90.000,E1 72.236} C_DIS
LIN {X -0.164,Y -577.918,Z 785.195,A 0.000,B 0.000,C 90.000,E1 71.148} C_DIS
LIN {X -0.099,Y -577.184,Z 785.186,A 0.000,B 0.000,C 90.000,E1 69.518} C_DIS
LIN {X -0.026,Y -576.477,Z 785.179,A 0.000,B 0.000,C 90.000,E1 68.156} C_DIS
LIN {X -0.118,Y -575.441,Z 785.170,A 0.000,B 0.000,C 90.000,E1 66.538} C_DIS
LIN {X -0.241,Y -574.211,Z 785.161,A 0.000,B 0.000,C 90.000,E1 64.921} C_DIS
LIN {X -0.104,Y -573.245,Z 785.155,A 0.000,B 0.000,C 90.000,E1 63.819} C_DIS
LIN {X -0.232,Y -572.090,Z 785.148,A 0.000,B 0.000,C 90.000,E1 62.743} C_DIS
LIN {X -0.118,Y -570.712,Z 785.142,A 0.000,B 0.000,C 90.000,E1 61.641} C_DIS
LIN {X 0.145,Y -569.557,Z 785.138,A 0.000,B 0.000,C 90.000,E1 60.795} C_DIS
LIN {X -0.280,Y -567.817,Z 785.132,A 0.000,B 0.000,C 90.000,E1 59.744} C_DIS
LIN {X 0.045,Y -565.804,Z 785.126,A 0.000,B 0.000,C 90.000,E1 58.614} C_DIS
LIN {X 0.056,Y -564.146,Z 785.121,A 0.000,B 0.000,C 90.000,E1 57.788} C_DIS
LIN {X 0.055,Y -562.250,Z 785.117,A 0.000,B 0.000,C 90.000,E1 56.962} C_DIS
LIN {X -0.183,Y -559.373,Z 785.110,A 0.000,B 0.000,C 90.000,E1 55.881} C_DIS
LIN {X -0.004,Y -557.850,Z 785.107,A 0.000,B 0.000,C 90.000,E1 55.308} C_DIS
LIN {X -0.072,Y -555.270,Z 785.103,A 0.000,B 0.000,C 90.000,E1 54.482} C_DIS
LIN {X 0.153,Y -552.483,Z 785.098,A 0.000,B 0.000,C 90.000,E1 53.623} C_DIS
LIN {X 0.016,Y -549.392,Z 785.093,A 0.000,B 0.000,C 90.000,E1 52.798} C_DIS
LIN {X -0.260,Y -545.895,Z 785.089,A 0.000,B 0.000,C 90.000,E1 51.984} C_DIS
LIN {X 0.163,Y -543.397,Z 785.086,A 0.000,B 0.000,C 90.000,E1 51.376} C_DIS
LIN {X 0.062,Y -539.988,Z 785.082,A 0.000,B 0.000,C 90.000,E1 50.678} C_DIS
LIN {X -0.154,Y -537.854,Z 785.079,A 0.000,B 0.000,C 90.000,E1 50.275} C_DIS
LIN {X 0.032,Y -533.775,Z 785.075,A 0.000,B 0.000,C 90.000,E1 49.542} C_DIS
LIN {X -0.041,Y -530.190,Z 785.072,A 0.000,B 0.000,C 90.000,E1 48.976} C_DIS
LIN {X -0.088,Y -526.215,Z 785.069,A 0.000,B 0.000,C 90.000,E1 48.405} C_DIS
LIN {X 0.179,Y -521.702,Z 785.066,A 0.000,B 0.000,C 90.000,E1 47.796} C_DIS
LIN {X 0.094,Y -516.851,Z 785.063,A 0.000,B 0.000,C 90.000,E1 47.229} C_DIS
LIN {X -0.094,Y -513.073,Z 785.060,A 0.000,B 0.000,C 90.000,E1 46.824} C_DIS
LIN {X 0.259,Y -507.487,Z 785.057,A 0.000,B 0.000,C 90.000,E1 46.215} C_DIS
LIN {X -0.090,Y -501.914,Z 785.054,A 0.000,B 0.000,C 90.000,E1 45.729} C_DIS
LIN {X -0.024,Y -492.957,Z 785.050,A 0.000,B 0.000,C 90.000,E1 44.960} C_DIS
LIN {X 0.004,Y -483.538,Z 785.046,A 0.000,B 0.000,C 90.000,E1 44.231} C_DIS
LIN {X -0.067,Y -477.194,Z 785.043,A 0.000,B 0.000,C 90.000,E1 43.785} C_DIS
LIN {X -0.178,Y -464.629,Z 785.038,A 0.000,B 0.000,C 90.000,E1 42.933} C_DIS
LIN {X -0.133,Y -448.507,Z 785.032,A 0.000,B 0.000,C 90.000,E1 41.838} C_DIS
LIN {X 0.050,Y -421.390,Z 785.021,A 0.000,B 0.000,C 90.000,E1 39.850} C_DIS
LIN {X -0.010,Y -412.272,Z 785.017,A 0.000,B 0.000,C 90.000,E1 39.116} C_DIS
LIN {X 0.008,Y -406.235,Z 785.014,A 0.000,B 0.000,C 90.000,E1 38.543} C_DIS
LIN {X -0.223,Y -405.926,Z 785.014,A 0.000,B 0.000,C 90.000,E1 38.543} C_DIS
LIN {X 0.001,Y -405.903,Z 785.014,A 0.000,B 0.000,C 90.000,E1 38.508} C_DIS
LIN {X 0.092,Y -397.537,Z 784.991,A 0.000,B 0.000,C 90.000,E1 34.278} C_DIS
LIN {X -0.148,Y -396.665,Z 784.988,A 0.000,B 0.000,C 90.000,E1 33.785} C_DIS
LIN {X 0.065,Y -396.503,Z 784.987,A 0.000,B 0.000,C 90.000,E1 33.579} C_DIS
LIN {X -0.035,Y -397.282,Z 784.970,A 0.000,B 0.000,C 90.000,E1 30.590} C_DIS
LIN {X 0.015,Y -398.636,Z 784.954,A 0.000,B 0.000,C 90.000,E1 27.769} C_DIS
LIN {X -0.147,Y -400.046,Z 784.941,A 0.000,B 0.000,C 90.000,E1 25.335} C_DIS
LIN {X -0.002,Y -401.989,Z 784.925,A 0.000,B 0.000,C 90.000,E1 22.514} C_DIS
LIN {X 0.135,Y -404.462,Z 784.910,A 0.000,B 0.000,C 90.000,E1 19.704} C_DIS
LIN {X 0.066,Y -409.502,Z 784.886,A 0.000,B 0.000,C 90.000,E1 15.552} C_DIS
LIN {X -0.148,Y -413.688,Z 784.871,A 0.000,B 0.000,C 90.000,E1 12.827} C_DIS
LIN {X -0.074,Y -417.734,Z 784.858,A 0.000,B 0.000,C 90.000,E1 10.423} C_DIS
LIN {X 0.165,Y -420.708,Z 784.848,A 0.000,B 0.000,C 90.000,E1 8.690} C_DIS
LIN {X 0.115,Y -423.675,Z 784.839,A 0.000,B 0.000,C 90.000,E1 7.004} C_DIS
LIN {X 0.143,Y -427.877,Z 784.826,A 0.000,B 0.000,C 90.000,E1 4.645} C_DIS
LIN {X 0.156,Y -431.595,Z 784.815,A 0.000,B 0.000,C 90.000,E1 2.636} C_DIS
LIN {X -0.191,Y -435.530,Z 784.804,A 0.000,B 0.000,C 90.000,E1 0.688} C_DIS
LIN {X -0.162,Y -440.789,Z 784.790,A 0.000,B 0.000,C 90.000,E1 358.165} C_DIS
LIN {X 0.164,Y -447.540,Z 784.773,A 0.000,B 0.000,C 90.000,E1 355.179} C_DIS
LIN {X 0.054,Y -451.360,Z 784.764,A 0.000,B 0.000,C 90.000,E1 353.571} C_DIS
LIN {X 0.115,Y -455.206,Z 784.755,A 0.000,B 0.000,C 90.000,E1 351.951} C_DIS
LIN {X -0.200,Y -458.944,Z 784.747,A 0.000,B 0.000,C 90.000,E1 350.387} C_DIS
LIN {X -0.126,Y -463.426,Z 784.736,A 0.000,B 0.000,C 90.000,E1 348.465} C_DIS
LIN {X 0.123,Y -464.219,Z 784.734,A 0.000,B 0.000,C 90.000,E1 348.117} C_DIS
LIN {X -0.182,Y -466.166,Z 784.731,A 0.000,B 0.000,C 90.000,E1 347.521} C_DIS
LIN {X 0.262,Y -467.994,Z 784.728,A 0.000,B 0.000,C 90.000,E1 346.992} C_DIS
LIN {X 0.074,Y -469.550,Z 784.726,A 0.000,B 0.000,C 90.000,E1 346.700} C_DIS
LIN {X -0.209,Y -472.939,Z 784.723,A 0.000,B 0.000,C 90.000,E1 346.228} C_DIS
LIN {X 0.002,Y -476.099,Z 784.721,A 0.000,B 0.000,C 90.000,E1 345.825} C_DIS
LIN {X 0.125,Y -482.126,Z 784.718,A 0.000,B 0.000,C 90.000,E1 345.227} C_DIS
LIN {X -0.049,Y -493.236,Z 784.713,A 0.000,B 0.000,C 90.000,E1 344.393} C_DIS
LIN {X -0.166,Y -518.433,Z 784.704,A 0.000,B 0.000,C 90.000,E1 342.670} C_DIS
LIN {X -0.288,Y -532.484,Z 784.699,A 0.000,B 0.000,C 90.000,E1 341.764} C_DIS
LIN {X -0.036,Y -540.161,Z 784.696,A 0.000,B 0.000,C 90.000,E1 341.221} C_DIS
LIN {X 0.052,Y -547.729,Z 784.693,A 0.000,B 0.000,C 90.000,E1 340.678} C_DIS
LIN {X -0.009,Y -553.599,Z 784.690,A 0.000,B 0.000,C 90.000,E1 340.242} C_DIS
LIN {X 0.270,Y -558.993,Z 784.688,A 0.000,B 0.000,C 90.000,E1 339.752} C_DIS
LIN {X -0.103,Y -564.034,Z 784.685,A 0.000,B 0.000,C 90.000,E1 339.316} C_DIS
LIN {X 0.166,Y -569.016,Z 784.682,A 0.000,B 0.000,C 90.000,E1 338.773} C_DIS
LIN {X 0.180,Y -573.790,Z 784.679,A 0.000,B 0.000,C 90.000,E1 338.230} C_DIS
LIN {X -0.154,Y -578.272,Z 784.676,A 0.000,B 0.000,C 90.000,E1 337.720} C_DIS
LIN {X -0.142,Y -582.551,Z 784.673,A 0.000,B 0.000,C 90.000,E1 337.177} C_DIS
LIN {X -0.001,Y -588.607,Z 784.669,A 0.000,B 0.000,C 90.000,E1 336.357} C_DIS
LIN {X 0.117,Y -595.985,Z 784.663,A 0.000,B 0.000,C 90.000,E1 335.281} C_DIS
LIN {X 0.080,Y -603.013,Z 784.657,A 0.000,B 0.000,C 90.000,E1 334.229} C_DIS
LIN {X -0.129,Y -608.820,Z 784.652,A 0.000,B 0.000,C 90.000,E1 333.332} C_DIS
LIN {X 0.026,Y -613.570,Z 784.648,A 0.000,B 0.000,C 90.000,E1 332.538} C_DIS
LIN {X -0.059,Y -618.836,Z 784.642,A 0.000,B 0.000,C 90.000,E1 331.641} C_DIS
LIN {X 0.215,Y -624.555,Z 784.637,A 0.000,B 0.000,C 90.000,E1 330.589} C_DIS
LIN {X 0.057,Y -632.049,Z 784.629,A 0.000,B 0.000,C 90.000,E1 329.203} C_DIS
LIN {X -0.055,Y -636.445,Z 784.624,A 0.000,B 0.000,C 90.000,E1 328.329} C_DIS
LIN {X -0.099,Y -641.152,Z 784.618,A 0.000,B 0.000,C 90.000,E1 327.327} C_DIS
LIN {X -0.148,Y -644.537,Z 784.614,A 0.000,B 0.000,C 90.000,E1 326.580} C_DIS
LIN {X 0.149,Y -649.717,Z 784.607,A 0.000,B 0.000,C 90.000,E1 325.308} C_DIS
LIN {X 0.097,Y -653.585,Z 784.602,A 0.000,B 0.000,C 90.000,E1 324.322} C_DIS
LIN {X 0.094,Y -657.163,Z 784.596,A 0.000,B 0.000,C 90.000,E1 323.336} C_DIS
LIN {X 0.086,Y -661.353,Z 784.590,A 0.000,B 0.000,C 90.000,E1 322.110} C_DIS
LIN {X -0.351,Y -664.449,Z 784.584,A 0.000,B 0.000,C 90.000,E1 321.170} C_DIS
LIN {X 0.169,Y -668.089,Z 784.577,A 0.000,B 0.000,C 90.000,E1 319.908} C_DIS
LIN {X 0.242,Y -671.473,Z 784.571,A 0.000,B 0.000,C 90.000,E1 318.690} C_DIS
LIN {X 0.369,Y -674.628,Z 784.564,A 0.000,B 0.000,C 90.000,E1 317.472} C_DIS
LIN {X 0.043,Y -677.285,Z 784.557,A 0.000,B 0.000,C 90.000,E1 316.296} C_DIS
LIN {X 0.271,Y -680.037,Z 784.549,A 0.000,B 0.000,C 90.000,E1 314.838} C_DIS
LIN {X 0.407,Y -681.364,Z 784.545,A 0.000,B 0.000,C 90.000,E1 314.109} C_DIS
LIN {X 0.239,Y -683.675,Z 784.537,A 0.000,B 0.000,C 90.000,E1 312.690} C_DIS
LIN {X -0.005,Y -685.122,Z 784.532,A 0.000,B 0.000,C 90.000,E1 311.757} C_DIS
LIN {X 0.340,Y -686.743,Z 784.525,A 0.000,B 0.000,C 90.000,E1 310.539} C_DIS
LIN {X 0.270,Y -688.106,Z 784.519,A 0.000,B 0.000,C 90.000,E1 309.358} C_DIS
LIN {X -0.373,Y -689.071,Z 784.514,A 0.000,B 0.000,C 90.000,E1 308.463} C_DIS
LIN {X 0.184,Y -690.514,Z 784.506,A 0.000,B 0.000,C 90.000,E1 306.996} C_DIS
LIN {X -0.062,Y -691.760,Z 784.498,A 0.000,B 0.000,C 90.000,E1 305.598} C_DIS
LIN {X -0.275,Y -692.872,Z 784.490,A 0.000,B 0.000,C 90.000,E1 304.199} C_DIS
LIN {X -0.016,Y -694.235,Z 784.479,A 0.000,B 0.000,C 90.000,E1 302.291} C_DIS
LIN {X 0.020,Y -695.350,Z 784.472,A 0.000,B 0.000,C 90.000,E1 300.875} C_DIS
LIN {X 0.165,Y -695.985,Z 784.466,A 0.000,B 0.000,C 90.000,E1 299.922} C_DIS
LIN {X 0.116,Y -696.814,Z 784.457,A 0.000,B 0.000,C 90.000,E1 298.281} C_DIS
LIN {X 0.378,Y -697.622,Z 784.448,A 0.000,B 0.000,C 90.000,E1 296.616} C_DIS
LIN {X -0.002,Y -698.835,Z 784.438,A 0.000,B 0.000,C 90.000,E1 294.771} C_DIS
LIN {X -0.398,Y -698.830,Z 784.435,A 0.000,B 0.000,C 90.000,E1 294.335} C_DIS
LIN {X -0.132,Y -698.673,Z 784.434,A 0.000,B 0.000,C 90.000,E1 294.079} C_DIS
LIN {X 0.112,Y -697.678,Z 784.431,A 0.000,B 0.000,C 90.000,E1 293.590} C_DIS
LIN {X -0.266,Y -696.837,Z 784.430,A 0.000,B 0.000,C 90.000,E1 293.387} C_DIS
LIN {X -0.156,Y -694.199,Z 784.428,A 0.000,B 0.000,C 90.000,E1 293.025} C_DIS
LIN {X 0.091,Y -692.098,Z 784.427,A 0.000,B 0.000,C 90.000,E1 292.770} C_DIS
LIN {X 0.213,Y -690.660,Z 784.426,A 0.000,B 0.000,C 90.000,E1 292.642} C_DIS
LIN {X -0.179,Y -688.576,Z 784.425,A 0.000,B 0.000,C 90.000,E1 292.567} C_DIS
LIN {X 0.238,Y -682.619,Z 784.424,A 0.000,B 0.000,C 90.000,E1 292.280} C_DIS
LIN {X 0.350,Y -680.690,Z 784.424,A 0.000,B 0.000,C 90.000,E1 292.206} C_DIS
LIN {X -0.020,Y -674.683,Z 784.423,A 0.000,B 0.000,C 90.000,E1 292.078} C_DIS
LIN {X 0.139,Y -669.399,Z 784.422,A 0.000,B 0.000,C 90.000,E1 291.972} C_DIS
LIN {X -0.048,Y -655.554,Z 784.421,A 0.000,B 0.000,C 90.000,E1 291.770} C_DIS
LIN {X -0.207,Y -637.955,Z 784.419,A 0.000,B 0.000,C 90.000,E1 291.461} C_DIS
LIN {X 0.154,Y -617.196,Z 784.417,A 0.000,B 0.000,C 90.000,E1 290.972} C_DIS
LIN {X -0.012,Y -599.888,Z 784.414,A 0.000,B 0.000,C 90.000,E1 290.556} C_DIS
LIN {X -0.029,Y -586.390,Z 784.412,A 0.000,B 0.000,C 90.000,E1 290.174} C_DIS
LIN {X -0.124,Y -572.829,Z 784.410,A 0.000,B 0.000,C 90.000,E1 289.758} C_DIS
LIN {X 0.121,Y -565.046,Z 784.408,A 0.000,B 0.000,C 90.000,E1 289.450} C_DIS
LIN {X 0.061,Y -561.374,Z 784.407,A 0.000,B 0.000,C 90.000,E1 289.268} C_DIS
LIN {X -0.111,Y -557.927,Z 784.406,A 0.000,B 0.000,C 90.000,E1 289.014} C_DIS
LIN {X -0.146,Y -556.928,Z 784.405,A 0.000,B 0.000,C 90.000,E1 288.852} C_DIS
LIN {X -0.261,Y -556.312,Z 784.404,A 0.000,B 0.000,C 90.000,E1 288.725} C_DIS
LIN {X 0.027,Y -555.505,Z 784.402,A 0.000,B 0.000,C 90.000,E1 288.417} C_DIS
LIN {X -0.147,Y -554.891,Z 784.400,A 0.000,B 0.000,C 90.000,E1 288.055} C_DIS
LIN {X 0.245,Y -554.401,Z 784.397,A 0.000,B 0.000,C 90.000,E1 287.457} C_DIS
LIN {X 0.218,Y -554.009,Z 784.393,A 0.000,B 0.000,C 90.000,E1 286.622} C_DIS
LIN {X 0.112,Y -552.995,Z 784.379,A 0.000,B 0.000,C 90.000,E1 284.120} C_DIS
LIN {X -0.244,Y -552.468,Z 784.369,A 0.000,B 0.000,C 90.000,E1 282.479} C_DIS
LIN {X 0.056,Y -551.820,Z 784.358,A 0.000,B 0.000,C 90.000,E1 280.489} C_DIS
LIN {X 0.005,Y -551.397,Z 784.351,A 0.000,B 0.000,C 90.000,E1 279.095} C_DIS
LIN {X 0.050,Y -551.032,Z 784.341,A 0.000,B 0.000,C 90.000,E1 277.409} C_DIS
LIN {X 0.236,Y -550.703,Z 784.337,A 0.000,B 0.000,C 90.000,E1 276.549} C_DIS
LIN {X 0.125,Y -549.808,Z 784.327,A 0.000,B 0.000,C 90.000,E1 274.878} C_DIS
LIN {X -0.053,Y -548.660,Z 784.318,A 0.000,B 0.000,C 90.000,E1 273.212} C_DIS
LIN {X -0.268,Y -547.624,Z 784.308,A 0.000,B 0.000,C 90.000,E1 271.547} C_DIS
LIN {X -0.037,Y -546.763,Z 784.301,A 0.000,B 0.000,C 90.000,E1 270.115} C_DIS
LIN {X 0.178,Y -545.759,Z 784.293,A 0.000,B 0.000,C 90.000,E1 268.682} C_DIS
LIN {X -0.063,Y -544.416,Z 784.282,A 0.000,B 0.000,C 90.000,E1 266.731} C_DIS
LIN {X 0.117,Y -543.597,Z 784.274,A 0.000,B 0.000,C 90.000,E1 265.298} C_DIS
LIN {X -0.170,Y -542.686,Z 784.266,A 0.000,B 0.000,C 90.000,E1 263.913} C_DIS
LIN {X 0.074,Y -541.578,Z 784.258,A 0.000,B 0.000,C 90.000,E1 262.470} C_DIS
LIN {X -0.097,Y -539.894,Z 784.247,A 0.000,B 0.000,C 90.000,E1 260.500} C_DIS
LIN {X 0.094,Y -538.925,Z 784.241,A 0.000,B 0.000,C 90.000,E1 259.342} C_DIS
LIN {X -0.032,Y -537.303,Z 784.231,A 0.000,B 0.000,C 90.000,E1 257.645} C_DIS
LIN {X -0.129,Y -535.940,Z 784.223,A 0.000,B 0.000,C 90.000,E1 256.228} C_DIS
LIN {X -0.202,Y -534.105,Z 784.214,A 0.000,B 0.000,C 90.000,E1 254.519} C_DIS
LIN {X -0.003,Y -531.842,Z 784.203,A 0.000,B 0.000,C 90.000,E1 252.489} C_DIS
LIN {X 0.095,Y -530.139,Z 784.195,A 0.000,B 0.000,C 90.000,E1 251.040} C_DIS
LIN {X 0.157,Y -528.582,Z 784.188,A 0.000,B 0.000,C 90.000,E1 249.880} C_DIS
LIN {X 0.230,Y -525.684,Z 784.177,A 0.000,B 0.000,C 90.000,E1 247.847} C_DIS
LIN {X 0.269,Y -522.986,Z 784.167,A 0.000,B 0.000,C 90.000,E1 246.102} C_DIS
LIN {X 0.262,Y -521.677,Z 784.163,A 0.000,B 0.000,C 90.000,E1 245.229} C_DIS
LIN {X 0.278,Y -519.281,Z 784.154,A 0.000,B 0.000,C 90.000,E1 243.768} C_DIS
LIN {X 0.118,Y -517.361,Z 784.148,A 0.000,B 0.000,C 90.000,E1 242.615} C_DIS
LIN {X -0.189,Y -515.791,Z 784.143,A 0.000,B 0.000,C 90.000,E1 241.769} C_DIS
LIN {X 0.196,Y -513.032,Z 784.135,A 0.000,B 0.000,C 90.000,E1 240.255} C_DIS
LIN {X 0.087,Y -510.237,Z 784.127,A 0.000,B 0.000,C 90.000,E1 238.791} C_DIS
LIN {X 0.294,Y -507.812,Z 784.120,A 0.000,B 0.000,C 90.000,E1 237.582} C_DIS
LIN {X -0.182,Y -506.642,Z 784.117,A 0.000,B 0.000,C 90.000,E1 237.041} C_DIS
LIN {X 0.240,Y -504.049,Z 784.110,A 0.000,B 0.000,C 90.000,E1 235.801} C_DIS
LIN {X 0.208,Y -501.325,Z 784.104,A 0.000,B 0.000,C 90.000,E1 234.609} C_DIS
LIN {X 0.134,Y -498.403,Z 784.097,A 0.000,B 0.000,C 90.000,E1 233.417} C_DIS
LIN {X 0.173,Y -494.609,Z 784.089,A 0.000,B 0.000,C 90.000,E1 231.904} C_DIS
LIN {X -0.086,Y -490.127,Z 784.078,A 0.000,B 0.000,C 90.000,E1 230.114} C_DIS
LIN {X 0.020,Y -483.875,Z 784.063,A 0.000,B 0.000,C 90.000,E1 227.349} C_DIS
LIN {X 0.009,Y -480.582,Z 784.055,A 0.000,B 0.000,C 90.000,E1 225.810} C_DIS
LIN {X 0.059,Y -476.453,Z 784.044,A 0.000,B 0.000,C 90.000,E1 223.947} C_DIS
LIN {X -0.063,Y -473.074,Z 784.036,A 0.000,B 0.000,C 90.000,E1 222.405} C_DIS
LIN {X -0.093,Y -468.360,Z 784.023,A 0.000,B 0.000,C 90.000,E1 220.216} C_DIS
LIN {X 0.093,Y -464.416,Z 784.013,A 0.000,B 0.000,C 90.000,E1 218.302} C_DIS
LIN {X -0.098,Y -460.422,Z 784.002,A 0.000,B 0.000,C 90.000,E1 216.423} C_DIS
LIN {X -0.174,Y -455.804,Z 783.990,A 0.000,B 0.000,C 90.000,E1 214.199} C_DIS
LIN {X -0.086,Y -451.897,Z 783.979,A 0.000,B 0.000,C 90.000,E1 212.260} C_DIS
LIN {X -0.189,Y -448.166,Z 783.968,A 0.000,B 0.000,C 90.000,E1 210.335} C_DIS
LIN {X -0.048,Y -445.029,Z 783.959,A 0.000,B 0.000,C 90.000,E1 208.693} C_DIS
LIN {X 0.023,Y -441.942,Z 783.950,A 0.000,B 0.000,C 90.000,E1 207.052} C_DIS
LIN {X 0.025,Y -438.804,Z 783.941,A 0.000,B 0.000,C 90.000,E1 205.412} C_DIS
LIN {X -0.021,Y -435.107,Z 783.930,A 0.000,B 0.000,C 90.000,E1 203.439} C_DIS
LIN {X -0.109,Y -431.278,Z 783.919,A 0.000,B 0.000,C 90.000,E1 201.461} C_DIS
LIN {X 0.140,Y -429.370,Z 783.914,A 0.000,B 0.000,C 90.000,E1 200.429} C_DIS
LIN {X -0.175,Y -424.883,Z 783.901,A 0.000,B 0.000,C 90.000,E1 198.127} C_DIS
LIN {X -0.165,Y -421.665,Z 783.891,A 0.000,B 0.000,C 90.000,E1 196.441} C_DIS
LIN {X 0.062,Y -418.305,Z 783.882,A 0.000,B 0.000,C 90.000,E1 194.717} C_DIS
LIN {X -0.106,Y -413.930,Z 783.869,A 0.000,B 0.000,C 90.000,E1 192.355} C_DIS
LIN {X 0.170,Y -410.733,Z 783.859,A 0.000,B 0.000,C 90.000,E1 190.602} C_DIS
LIN {X -0.045,Y -405.953,Z 783.844,A 0.000,B 0.000,C 90.000,E1 187.871} C_DIS
LIN {X -0.071,Y -404.223,Z 783.838,A 0.000,B 0.000,C 90.000,E1 186.834} C_DIS
LIN {X -0.184,Y -400.665,Z 783.826,A 0.000,B 0.000,C 90.000,E1 184.759} C_DIS
LIN {X -0.004,Y -394.551,Z 783.803,A 0.000,B 0.000,C 90.000,E1 180.516} C_DIS
LIN {X 0.043,Y -392.534,Z 783.793,A 0.000,B 0.000,C 90.000,E1 178.740} C_DIS
LIN {X -0.099,Y -389.953,Z 783.779,A 0.000,B 0.000,C 90.000,E1 176.274} C_DIS
LIN {X -0.087,Y -388.230,Z 783.769,A 0.000,B 0.000,C 90.000,E1 174.489} C_DIS
LIN {X 0.137,Y -385.842,Z 783.755,A 0.000,B 0.000,C 90.000,E1 171.951} C_DIS
LIN {X -0.140,Y -383.163,Z 783.737,A 0.000,B 0.000,C 90.000,E1 168.757} C_DIS
LIN {X 0.163,Y -381.119,Z 783.719,A 0.000,B 0.000,C 90.000,E1 165.463} C_DIS
LIN {X -0.042,Y -379.880,Z 783.705,A 0.000,B 0.000,C 90.000,E1 162.960} C_DIS
LIN {X -0.057,Y -378.965,Z 783.689,A 0.000,B 0.000,C 90.000,E1 160.061} C_DIS
LIN {X -0.127,Y -379.135,Z 783.655,A 0.000,B 0.000,C 90.000,E1 153.896} C_DIS
LIN {X 0.056,Y -380.114,Z 783.643,A 0.000,B 0.000,C 90.000,E1 151.691} C_DIS
LIN {X 0.116,Y -381.534,Z 783.633,A 0.000,B 0.000,C 90.000,E1 149.871} C_DIS
LIN {X 0.088,Y -384.152,Z 783.621,A 0.000,B 0.000,C 90.000,E1 147.709} C_DIS
LIN {X -0.192,Y -388.130,Z 783.609,A 0.000,B 0.000,C 90.000,E1 145.595} C_DIS
LIN {X 0.019,Y -389.828,Z 783.605,A 0.000,B 0.000,C 90.000,E1 144.848} C_DIS
LIN {X -0.202,Y -392.589,Z 783.600,A 0.000,B 0.000,C 90.000,E1 143.989} C_DIS
LIN {X -0.042,Y -395.253,Z 783.596,A 0.000,B 0.000,C 90.000,E1 143.256} C_DIS
LIN {X 0.016,Y -397.562,Z 783.593,A 0.000,B 0.000,C 90.000,E1 142.718} C_DIS
LIN {X -0.091,Y -401.295,Z 783.589,A 0.000,B 0.000,C 90.000,E1 142.029} C_DIS
LIN {X -0.092,Y -404.323,Z 783.586,A 0.000,B 0.000,C 90.000,E1 141.537} C_DIS
LIN {X 0.121,Y -408.830,Z 783.583,A 0.000,B 0.000,C 90.000,E1 140.884} C_DIS
LIN {X -0.170,Y -428.302,Z 783.570,A 0.000,B 0.000,C 90.000,E1 138.609} C_DIS
LIN {X 0.181,Y -437.995,Z 783.564,A 0.000,B 0.000,C 90.000,E1 137.472} C_DIS
LIN {X -0.013,Y -450.508,Z 783.556,A 0.000,B 0.000,C 90.000,E1 136.095} C_DIS
LIN {X 0.088,Y -459.723,Z 783.550,A 0.000,B 0.000,C 90.000,E1 135.000} C_DIS
LIN {X 0.254,Y -465.970,Z 783.546,A 0.000,B 0.000,C 90.000,E1 134.190} C_DIS
LIN {X -0.164,Y -476.639,Z 783.538,A 0.000,B 0.000,C 90.000,E1 132.852} C_DIS
LIN {X -0.184,Y -482.324,Z 783.534,A 0.000,B 0.000,C 90.000,E1 132.081} C_DIS
LIN {X -0.106,Y -488.893,Z 783.529,A 0.000,B 0.000,C 90.000,E1 131.148} C_DIS
LIN {X -0.109,Y -496.956,Z 783.522,A 0.000,B 0.000,C 90.000,E1 129.930} C_DIS
LIN {X -0.292,Y -501.703,Z 783.518,A 0.000,B 0.000,C 90.000,E1 129.197} C_DIS
LIN {X -0.032,Y -508.787,Z 783.511,A 0.000,B 0.000,C 90.000,E1 127.971} C_DIS
LIN {X -0.102,Y -512.889,Z 783.507,A 0.000,B 0.000,C 90.000,E1 127.237} C_DIS
LIN {X 0.331,Y -519.117,Z 783.500,A 0.000,B 0.000,C 90.000,E1 126.011} C_DIS
LIN {X -0.176,Y -525.006,Z 783.494,A 0.000,B 0.000,C 90.000,E1 124.898} C_DIS
LIN {X -0.085,Y -526.995,Z 783.491,A 0.000,B 0.000,C 90.000,E1 124.452} C_DIS
LIN {X 0.144,Y -531.951,Z 783.485,A 0.000,B 0.000,C 90.000,E1 123.293} C_DIS
LIN {X 0.248,Y -536.547,Z 783.479,A 0.000,B 0.000,C 90.000,E1 122.133} C_DIS
LIN {X 0.134,Y -540.957,Z 783.472,A 0.000,B 0.000,C 90.000,E1 121.003} C_DIS
LIN {X 0.347,Y -543.970,Z 783.468,A 0.000,B 0.000,C 90.000,E1 120.129} C_DIS
LIN {X 0.071,Y -547.696,Z 783.461,A 0.000,B 0.000,C 90.000,E1 119.027} C_DIS
LIN {X 0.090,Y -550.356,Z 783.457,A 0.000,B 0.000,C 90.000,E1 118.180} C_DIS
LIN {X 0.137,Y -552.862,Z 783.452,A 0.000,B 0.000,C 90.000,E1 117.334} C_DIS
LIN {X 0.207,Y -555.002,Z 783.447,A 0.000,B 0.000,C 90.000,E1 116.488} C_DIS
LIN {X 0.051,Y -556.790,Z 783.443,A 0.000,B 0.000,C 90.000,E1 115.668} C_DIS
LIN {X -0.083,Y -558.309,Z 783.438,A 0.000,B 0.000,C 90.000,E1 114.847} C_DIS
LIN {X 0.027,Y -559.492,Z 783.433,A 0.000,B 0.000,C 90.000,E1 114.003} C_DIS
LIN {X 0.104,Y -561.303,Z 783.424,A 0.000,B 0.000,C 90.000,E1 112.333} C_DIS
LIN {X 0.113,Y -562.529,Z 783.418,A 0.000,B 0.000,C 90.000,E1 111.227} C_DIS
LIN {X -0.070,Y -563.801,Z 783.410,A 0.000,B 0.000,C 90.000,E1 109.866} C_DIS
LIN {X -0.081,Y -564.924,Z 783.403,A 0.000,B 0.000,C 90.000,E1 108.489} C_DIS
LIN {X -0.275,Y -566.088,Z 783.394,A 0.000,B 0.000,C 90.000,E1 106.858} C_DIS
LIN {X -0.071,Y -567.239,Z 783.384,A 0.000,B 0.000,C 90.000,E1 105.190} C_DIS
LIN {X -0.181,Y -568.947,Z 783.372,A 0.000,B 0.000,C 90.000,E1 103.008} C_DIS
LIN {X 0.001,Y -570.516,Z 783.362,A 0.000,B 0.000,C 90.000,E1 101.074} C_DIS
LIN {X 0.199,Y -571.411,Z 783.356,A 0.000,B 0.000,C 90.000,E1 99.962} C_DIS
LIN {X 0.041,Y -572.795,Z 783.346,A 0.000,B 0.000,C 90.000,E1 98.341} C_DIS
LIN {X -0.209,Y -573.773,Z 783.339,A 0.000,B 0.000,C 90.000,E1 97.004} C_DIS
LIN {X -0.016,Y -574.679,Z 783.331,A 0.000,B 0.000,C 90.000,E1 95.625} C_DIS
LIN {X -0.044,Y -575.761,Z 783.321,A 0.000,B 0.000,C 90.000,E1 93.726} C_DIS
LIN {X 0.154,Y -576.468,Z 783.313,A 0.000,B 0.000,C 90.000,E1 92.350} C_DIS
LIN {X -0.211,Y -577.111,Z 783.306,A 0.000,B 0.000,C 90.000,E1 91.031} C_DIS
LIN {X 0.156,Y -577.803,Z 783.297,A 0.000,B 0.000,C 90.000,E1 89.370} C_DIS
LIN {X -0.027,Y -578.374,Z 783.288,A 0.000,B 0.000,C 90.000,E1 87.764} C_DIS
LIN {X -0.202,Y -578.787,Z 783.279,A 0.000,B 0.000,C 90.000,E1 86.159} C_DIS
LIN {X -0.070,Y -579.050,Z 783.273,A 0.000,B 0.000,C 90.000,E1 85.065} C_DIS
LIN {X 0.004,Y -579.344,Z 783.262,A 0.000,B 0.000,C 90.000,E1 83.166} C_DIS
LIN {X -0.215,Y -579.594,Z 783.255,A 0.000,B 0.000,C 90.000,E1 81.837} C_DIS
LIN {X 0.231,Y -579.696,Z 783.247,A 0.000,B 0.000,C 90.000,E1 80.443} C_DIS
LIN {X 0.107,Y -579.835,Z 783.240,A 0.000,B 0.000,C 90.000,E1 79.106} C_DIS
LIN {X -0.129,Y -579.817,Z 783.234,A 0.000,B 0.000,C 90.000,E1 78.049} C_DIS
LIN {X -0.137,Y -579.676,Z 783.226,A 0.000,B 0.000,C 90.000,E1 76.700} C_DIS
LIN {X -0.138,Y -579.309,Z 783.216,A 0.000,B 0.000,C 90.000,E1 74.810} C_DIS
LIN {X -0.004,Y -578.815,Z 783.205,A 0.000,B 0.000,C 90.000,E1 72.906} C_DIS
LIN {X 0.081,Y -578.228,Z 783.196,A 0.000,B 0.000,C 90.000,E1 71.275} C_DIS
LIN {X 0.149,Y -577.457,Z 783.187,A 0.000,B 0.000,C 90.000,E1 69.645} C_DIS
LIN {X 0.066,Y -576.581,Z 783.178,A 0.000,B 0.000,C 90.000,E1 68.028} C_DIS
LIN {X -0.022,Y -575.501,Z 783.169,A 0.000,B 0.000,C 90.000,E1 66.410} C_DIS
LIN {X -0.143,Y -574.233,Z 783.160,A 0.000,B 0.000,C 90.000,E1 64.793} C_DIS
LIN {X -0.005,Y -573.204,Z 783.154,A 0.000,B 0.000,C 90.000,E1 63.691} C_DIS
LIN {X 0.028,Y -572.307,Z 783.149,A 0.000,B 0.000,C 90.000,E1 62.871} C_DIS
LIN {X -0.024,Y -570.546,Z 783.142,A 0.000,B 0.000,C 90.000,E1 61.513} C_DIS
LIN {X 0.238,Y -569.334,Z 783.137,A 0.000,B 0.000,C 90.000,E1 60.667} C_DIS
LIN {X 0.096,Y -567.550,Z 783.131,A 0.000,B 0.000,C 90.000,E1 59.587} C_DIS
LIN {X -0.167,Y -566.022,Z 783.127,A 0.000,B 0.000,C 90.000,E1 58.791} C_DIS
LIN {X 0.132,Y -563.702,Z 783.120,A 0.000,B 0.000,C 90.000,E1 57.661} C_DIS
LIN {X 0.125,Y -561.758,Z 783.116,A 0.000,B 0.000,C 90.000,E1 56.834} C_DIS
LIN {X -0.124,Y -558.785,Z 783.110,A 0.000,B 0.000,C 90.000,E1 55.754} C_DIS
LIN {X 0.134,Y -556.312,Z 783.105,A 0.000,B 0.000,C 90.000,E1 54.895} C_DIS
LIN {X 0.117,Y -552.689,Z 783.099,A 0.000,B 0.000,C 90.000,E1 53.783} C_DIS
LIN {X -0.128,Y -549.594,Z 783.094,A 0.000,B 0.000,C 90.000,E1 52.970} C_DIS
LIN {X -0.155,Y -546.700,Z 783.090,A 0.000,B 0.000,C 90.000,E1 52.271} C_DIS
LIN {X 0.123,Y -543.575,Z 783.086,A 0.000,B 0.000,C 90.000,E1 51.537} C_DIS
LIN {X -0.055,Y -540.141,Z 783.083,A 0.000,B 0.000,C 90.000,E1 50.848} C_DIS
LIN {X -0.019,Y -537.246,Z 783.079,A 0.000,B 0.000,C 90.000,E1 50.275} C_DIS
LIN {X 0.163,Y -533.068,Z 783.075,A 0.000,B 0.000,C 90.000,E1 49.542} C_DIS
LIN {X -0.264,Y -529.397,Z 783.072,A 0.000,B 0.000,C 90.000,E1 49.013} C_DIS
LIN {X 0.031,Y -525.327,Z 783.069,A 0.000,B 0.000,C 90.000,E1 48.405} C_DIS
LIN {X -0.096,Y -520.686,Z 783.066,A 0.000,B 0.000,C 90.000,E1 47.838} C_DIS
LIN {X -0.010,Y -517.016,Z 783.063,A 0.000,B 0.000,C 90.000,E1 47.391} C_DIS
LIN {X -0.113,Y -511.751,Z 783.060,A 0.000,B 0.000,C 90.000,E1 46.824} C_DIS
LIN {X 0.017,Y -506.182,Z 783.057,A 0.000,B 0.000,C 90.000,E1 46.257} C_DIS
LIN {X -0.315,Y -501.856,Z 783.055,A 0.000,B 0.000,C 90.000,E1 45.891} C_DIS
LIN {X 0.158,Y -495.791,Z 783.052,A 0.000,B 0.000,C 90.000,E1 45.324} C_DIS
LIN {X -0.238,Y -491.248,Z 783.050,A 0.000,B 0.000,C 90.000,E1 45.000} C_DIS
LIN {X -0.094,Y -481.911,Z 783.046,A 0.000,B 0.000,C 90.000,E1 44.271} C_DIS
LIN {X 0.046,Y -472.183,Z 783.042,A 0.000,B 0.000,C 90.000,E1 43.581} C_DIS
LIN {X 0.191,Y -459.317,Z 783.037,A 0.000,B 0.000,C 90.000,E1 42.690} C_DIS
LIN {X 0.017,Y -439.983,Z 783.030,A 0.000,B 0.000,C 90.000,E1 41.391} C_DIS
LIN {X 0.129,Y -417.807,Z 783.021,A 0.000,B 0.000,C 90.000,E1 39.725} C_DIS
LIN {X 0.240,Y -411.710,Z 783.018,A 0.000,B 0.000,C 90.000,E1 39.197} C_DIS
LIN {X 0.041,Y -408.733,Z 783.016,A 0.000,B 0.000,C 90.000,E1 38.955} C_DIS
LIN {X -0.012,Y -406.234,Z 783.015,A 0.000,B 0.000,C 90.000,E1 38.705} C_DIS
LIN {X -0.038,Y -406.208,Z 783.015,A 0.000,B 0.000,C 90.000,E1 38.705} C_DIS
LIN {X 0.049,Y -404.548,Z 783.011,A 0.000,B 0.000,C 90.000,E1 37.890} C_DIS
LIN {X 0.085,Y -396.850,Z 782.988,A 0.000,B 0.000,C 90.000,E1 33.865} C_DIS
LIN {X -0.014,Y -396.846,Z 782.984,A 0.000,B 0.000,C 90.000,E1 33.166} C_DIS
LIN {X -0.166,Y -398.003,Z 782.965,A 0.000,B 0.000,C 90.000,E1 29.667} C_DIS
LIN {X 0.023,Y -399.217,Z 782.951,A 0.000,B 0.000,C 90.000,E1 27.180} C_DIS
LIN {X -0.002,Y -400.487,Z 782.939,A 0.000,B 0.000,C 90.000,E1 25.079} C_DIS
LIN {X -0.044,Y -403.084,Z 782.920,A 0.000,B 0.000,C 90.000,E1 21.589} C_DIS
LIN {X -0.063,Y -406.914,Z 782.899,A 0.000,B 0.000,C 90.000,E1 17.764} C_DIS
LIN {X 0.121,Y -409.660,Z 782.887,A 0.000,B 0.000,C 90.000,E1 15.662} C_DIS
LIN {X -0.096,Y -413.845,Z 782.872,A 0.000,B 0.000,C 90.000,E1 12.939} C_DIS
LIN {X -0.100,Y -417.863,Z 782.859,A 0.000,B 0.000,C 90.000,E1 10.546} C_DIS
LIN {X -0.133,Y -421.409,Z 782.847,A 0.000,B 0.000,C 90.000,E1 8.511} C_DIS
LIN {X -0.152,Y -424.948,Z 782.836,A 0.000,B 0.000,C 90.000,E1 6.486} C_DIS
LIN {X -0.182,Y -428.544,Z 782.825,A 0.000,B 0.000,C 90.000,E1 4.473} C_DIS
LIN {X 0.036,Y -430.414,Z 782.819,A 0.000,B 0.000,C 90.000,E1 3.440} C_DIS
LIN {X -0.144,Y -435.564,Z 782.804,A 0.000,B 0.000,C 90.000,E1 0.802} C_DIS
LIN {X -0.157,Y -441.052,Z 782.790,A 0.000,B 0.000,C 90.000,E1 358.165} C_DIS
LIN {X 0.179,Y -447.770,Z 782.773,A 0.000,B 0.000,C 90.000,E1 355.179} C_DIS
LIN {X 0.073,Y -451.590,Z 782.764,A 0.000,B 0.000,C 90.000,E1 353.571} C_DIS
LIN {X 0.138,Y -455.429,Z 782.755,A 0.000,B 0.000,C 90.000,E1 351.951} C_DIS
LIN {X -0.173,Y -459.149,Z 782.747,A 0.000,B 0.000,C 90.000,E1 350.387} C_DIS
LIN {X 0.051,Y -465.147,Z 782.732,A 0.000,B 0.000,C 90.000,E1 347.813} C_DIS
LIN {X 0.111,Y -467.160,Z 782.729,A 0.000,B 0.000,C 90.000,E1 347.173} C_DIS
LIN {X 0.104,Y -469.080,Z 782.726,A 0.000,B 0.000,C 90.000,E1 346.700} C_DIS
LIN {X -0.082,Y -470.679,Z 782.724,A 0.000,B 0.000,C 90.000,E1 346.408} C_DIS
LIN {X -0.070,Y -473.969,Z 782.722,A 0.000,B 0.000,C 90.000,E1 345.936} C_DIS
LIN {X 0.145,Y -477.344,Z 782.720,A 0.000,B 0.000,C 90.000,E1 345.519} C_DIS
LIN {X -0.231,Y -482.812,Z 782.717,A 0.000,B 0.000,C 90.000,E1 345.046} C_DIS
LIN {X 0.090,Y -494.685,Z 782.712,A 0.000,B 0.000,C 90.000,E1 344.102} C_DIS
LIN {X -0.060,Y -508.674,Z 782.706,A 0.000,B 0.000,C 90.000,E1 343.142} C_DIS
LIN {X 0.102,Y -529.214,Z 782.699,A 0.000,B 0.000,C 90.000,E1 341.764} C_DIS
LIN {X 0.128,Y -538.561,Z 782.695,A 0.000,B 0.000,C 90.000,E1 341.148} C_DIS
LIN {X 0.304,Y -546.158,Z 782.692,A 0.000,B 0.000,C 90.000,E1 340.604} C_DIS
LIN {X 0.101,Y -552.078,Z 782.690,A 0.000,B 0.000,C 90.000,E1 340.188} C_DIS
LIN {X -0.237,Y -557.685,Z 782.687,A 0.000,B 0.000,C 90.000,E1 339.752} C_DIS
LIN {X 0.254,Y -562.999,Z 782.685,A 0.000,B 0.000,C 90.000,E1 339.209} C_DIS
LIN {X -0.028,Y -568.046,Z 782.682,A 0.000,B 0.000,C 90.000,E1 338.720} C_DIS
LIN {X 0.221,Y -572.879,Z 782.679,A 0.000,B 0.000,C 90.000,E1 338.156} C_DIS
LIN {X 0.199,Y -577.437,Z 782.676,A 0.000,B 0.000,C 90.000,E1 337.614} C_DIS
LIN {X -0.108,Y -581.730,Z 782.673,A 0.000,B 0.000,C 90.000,E1 337.102} C_DIS
LIN {X -0.266,Y -588.860,Z 782.668,A 0.000,B 0.000,C 90.000,E1 336.177} C_DIS
LIN {X -0.152,Y -596.231,Z 782.662,A 0.000,B 0.000,C 90.000,E1 335.101} C_DIS
LIN {X 0.070,Y -603.267,Z 782.656,A 0.000,B 0.000,C 90.000,E1 334.024} C_DIS
LIN {X -0.156,Y -609.885,Z 782.650,A 0.000,B 0.000,C 90.000,E1 332.999} C_DIS
LIN {X -0.271,Y -614.610,Z 782.646,A 0.000,B 0.000,C 90.000,E1 332.231} C_DIS
LIN {X -0.047,Y -619.079,Z 782.641,A 0.000,B 0.000,C 90.000,E1 331.435} C_DIS
LIN {X -0.076,Y -624.134,Z 782.636,A 0.000,B 0.000,C 90.000,E1 330.539} C_DIS
LIN {X -0.268,Y -630.410,Z 782.630,A 0.000,B 0.000,C 90.000,E1 329.410} C_DIS
LIN {X 0.124,Y -634.339,Z 782.626,A 0.000,B 0.000,C 90.000,E1 328.614} C_DIS
LIN {X -0.003,Y -637.400,Z 782.622,A 0.000,B 0.000,C 90.000,E1 327.995} C_DIS
LIN {X -0.041,Y -642.072,Z 782.617,A 0.000,B 0.000,C 90.000,E1 326.993} C_DIS
LIN {X 0.277,Y -645.408,Z 782.612,A 0.000,B 0.000,C 90.000,E1 326.215} C_DIS
LIN {X -0.204,Y -649.540,Z 782.607,A 0.000,B 0.000,C 90.000,E1 325.261} C_DIS
LIN {X -0.267,Y -653.464,Z 782.601,A 0.000,B 0.000,C 90.000,E1 324.276} C_DIS
LIN {X 0.113,Y -657.066,Z 782.596,A 0.000,B 0.000,C 90.000,E1 323.256} C_DIS
LIN {X 0.106,Y -661.301,Z 782.589,A 0.000,B 0.000,C 90.000,E1 322.029} C_DIS
LIN {X -0.330,Y -664.444,Z 782.584,A 0.000,B 0.000,C 90.000,E1 321.090} C_DIS
LIN {X 0.192,Y -668.135,Z 782.577,A 0.000,B 0.000,C 90.000,E1 319.828} C_DIS
LIN {X 0.261,Y -670.890,Z 782.572,A 0.000,B 0.000,C 90.000,E1 318.852} C_DIS
LIN {X -0.121,Y -674.160,Z 782.565,A 0.000,B 0.000,C 90.000,E1 317.676} C_DIS
LIN {X 0.043,Y -676.904,Z 782.558,A 0.000,B 0.000,C 90.000,E1 316.458} C_DIS
LIN {X 0.263,Y -679.763,Z 782.550,A 0.000,B 0.000,C 90.000,E1 315.000} C_DIS
LIN {X 0.019,Y -681.945,Z 782.544,A 0.000,B 0.000,C 90.000,E1 313.824} C_DIS
LIN {X 0.279,Y -683.899,Z 782.537,A 0.000,B 0.000,C 90.000,E1 312.609} C_DIS
LIN {X 0.093,Y -685.686,Z 782.530,A 0.000,B 0.000,C 90.000,E1 311.434} C_DIS
LIN {X -0.003,Y -687.312,Z 782.524,A 0.000,B 0.000,C 90.000,E1 310.253} C_DIS
LIN {X -0.061,Y -688.644,Z 782.517,A 0.000,B 0.000,C 90.000,E1 309.072} C_DIS
LIN {X 0.133,Y -690.278,Z 782.508,A 0.000,B 0.000,C 90.000,E1 307.397} C_DIS
LIN {X -0.132,Y -690.969,Z 782.504,A 0.000,B 0.000,C 90.000,E1 306.710} C_DIS
LIN {X -0.368,Y -692.198,Z 782.496,A 0.000,B 0.000,C 90.000,E1 305.311} C_DIS
LIN {X -0.222,Y -693.127,Z 782.490,A 0.000,B 0.000,C 90.000,E1 304.119} C_DIS
LIN {X 0.038,Y -694.494,Z 782.479,A 0.000,B 0.000,C 90.000,E1 302.212} C_DIS
LIN {X 0.072,Y -695.589,Z 782.471,A 0.000,B 0.000,C 90.000,E1 300.797} C_DIS
LIN {X -0.131,Y -696.204,Z 782.466,A 0.000,B 0.000,C 90.000,E1 299.873} C_DIS
LIN {X 0.191,Y -696.894,Z 782.458,A 0.000,B 0.000,C 90.000,E1 298.437} C_DIS
LIN {X 0.161,Y -697.667,Z 782.449,A 0.000,B 0.000,C 90.000,E1 296.796} C_DIS
LIN {X 0.035,Y -698.984,Z 782.437,A 0.000,B 0.000,C 90.000,E1 294.695} C_DIS
LIN {X 0.276,Y -698.907,Z 782.435,A 0.000,B 0.000,C 90.000,E1 294.207} C_DIS
LIN {X -0.098,Y -698.620,Z 782.433,A 0.000,B 0.000,C 90.000,E1 294.003} C_DIS
LIN {X 0.146,Y -697.539,Z 782.431,A 0.000,B 0.000,C 90.000,E1 293.515} C_DIS
LIN {X 0.404,Y -696.397,Z 782.429,A 0.000,B 0.000,C 90.000,E1 293.259} C_DIS
LIN {X -0.254,Y -694.467,Z 782.428,A 0.000,B 0.000,C 90.000,E1 293.078} C_DIS
LIN {X -0.005,Y -692.361,Z 782.427,A 0.000,B 0.000,C 90.000,E1 292.823} C_DIS
LIN {X 0.115,Y -691.113,Z 782.426,A 0.000,B 0.000,C 90.000,E1 292.695} C_DIS
LIN {X -0.032,Y -689.144,Z 782.426,A 0.000,B 0.000,C 90.000,E1 292.589} C_DIS
LIN {X 0.072,Y -683.266,Z 782.424,A 0.000,B 0.000,C 90.000,E1 292.333} C_DIS
LIN {X 0.114,Y -679.329,Z 782.423,A 0.000,B 0.000,C 90.000,E1 292.206} C_DIS
LIN {X -0.131,Y -673.518,Z 782.423,A 0.000,B 0.000,C 90.000,E1 292.078} C_DIS
LIN {X -0.088,Y -654.089,Z 782.421,A 0.000,B 0.000,C 90.000,E1 291.770} C_DIS
LIN {X -0.286,Y -640.209,Z 782.420,A 0.000,B 0.000,C 90.000,E1 291.535} C_DIS
LIN {X 0.143,Y -619.433,Z 782.417,A 0.000,B 0.000,C 90.000,E1 291.046} C_DIS
LIN {X -0.132,Y -598.713,Z 782.414,A 0.000,B 0.000,C 90.000,E1 290.556} C_DIS
LIN {X -0.166,Y -585.293,Z 782.412,A 0.000,B 0.000,C 90.000,E1 290.174} C_DIS
LIN {X -0.098,Y -568.433,Z 782.409,A 0.000,B 0.000,C 90.000,E1 289.631} C_DIS
LIN {X 0.031,Y -565.371,Z 782.408,A 0.000,B 0.000,C 90.000,E1 289.504} C_DIS
LIN {X 0.009,Y -561.336,Z 782.407,A 0.000,B 0.000,C 90.000,E1 289.322} C_DIS
LIN {X -0.203,Y -558.158,Z 782.406,A 0.000,B 0.000,C 90.000,E1 289.087} C_DIS
LIN {X -0.156,Y -557.618,Z 782.406,A 0.000,B 0.000,C 90.000,E1 289.033} C_DIS
LIN {X -0.084,Y -556.631,Z 782.405,A 0.000,B 0.000,C 90.000,E1 288.833} C_DIS
LIN {X 0.147,Y -556.089,Z 782.404,A 0.000,B 0.000,C 90.000,E1 288.671} C_DIS
LIN {X 0.316,Y -555.186,Z 782.402,A 0.000,B 0.000,C 90.000,E1 288.236} C_DIS
LIN {X 0.182,Y -554.595,Z 782.398,A 0.000,B 0.000,C 90.000,E1 287.692} C_DIS
LIN {X 0.155,Y -554.268,Z 782.394,A 0.000,B 0.000,C 90.000,E1 286.858} C_DIS
LIN {X 0.214,Y -553.372,Z 782.383,A 0.000,B 0.000,C 90.000,E1 284.898} C_DIS
LIN {X 0.245,Y -552.700,Z 782.372,A 0.000,B 0.000,C 90.000,E1 282.939} C_DIS
LIN {X -0.122,Y -552.121,Z 782.363,A 0.000,B 0.000,C 90.000,E1 281.299} C_DIS
LIN {X -0.061,Y -551.599,Z 782.353,A 0.000,B 0.000,C 90.000,E1 279.613} C_DIS
LIN {X 0.129,Y -551.047,Z 782.341,A 0.000,B 0.000,C 90.000,E1 277.352} C_DIS
LIN {X -0.168,Y -550.708,Z 782.336,A 0.000,B 0.000,C 90.000,E1 276.543} C_DIS
LIN {X 0.160,Y -549.945,Z 782.328,A 0.000,B 0.000,C 90.000,E1 275.106} C_DIS
LIN {X -0.020,Y -548.827,Z 782.319,A 0.000,B 0.000,C 90.000,E1 273.440} C_DIS
LIN {X -0.186,Y -547.599,Z 782.308,A 0.000,B 0.000,C 90.000,E1 271.489} C_DIS
LIN {X -0.002,Y -546.942,Z 782.302,A 0.000,B 0.000,C 90.000,E1 270.344} C_DIS
LIN {X 0.258,Y -545.744,Z 782.293,A 0.000,B 0.000,C 90.000,E1 268.625} C_DIS
LIN {X 0.016,Y -544.385,Z 782.282,A 0.000,B 0.000,C 90.000,E1 266.674} C_DIS
LIN {X 0.263,Y -543.387,Z 782.272,A 0.000,B 0.000,C 90.000,E1 264.951} C_DIS
LIN {X -0.095,Y -542.667,Z 782.266,A 0.000,B 0.000,C 90.000,E1 263.856} C_DIS
LIN {X 0.148,Y -541.545,Z 782.258,A 0.000,B 0.000,C 90.000,E1 262.413} C_DIS
LIN {X -0.028,Y -539.853,Z 782.247,A 0.000,B 0.000,C 90.000,E1 260.443} C_DIS
LIN {X 0.229,Y -538.608,Z 782.239,A 0.000,B 0.000,C 90.000,E1 258.993} C_DIS
LIN {X 0.031,Y -537.292,Z 782.231,A 0.000,B 0.000,C 90.000,E1 257.589} C_DIS
LIN {X -0.070,Y -535.925,Z 782.223,A 0.000,B 0.000,C 90.000,E1 256.172} C_DIS
LIN {X -0.003,Y -534.111,Z 782.214,A 0.000,B 0.000,C 90.000,E1 254.448} C_DIS
LIN {X -0.272,Y -531.496,Z 782.201,A 0.000,B 0.000,C 90.000,E1 252.181} C_DIS
LIN {X -0.175,Y -529.759,Z 782.193,A 0.000,B 0.000,C 90.000,E1 250.732} C_DIS
LIN {X 0.197,Y -528.568,Z 782.188,A 0.000,B 0.000,C 90.000,E1 249.826} C_DIS
LIN {X 0.091,Y -526.074,Z 782.178,A 0.000,B 0.000,C 90.000,E1 248.103} C_DIS
LIN {X -0.029,Y -523.859,Z 782.170,A 0.000,B 0.000,C 90.000,E1 246.666} C_DIS
LIN {X -0.188,Y -521.653,Z 782.162,A 0.000,B 0.000,C 90.000,E1 245.229} C_DIS
LIN {X -0.033,Y -518.781,Z 782.153,A 0.000,B 0.000,C 90.000,E1 243.461} C_DIS
LIN {X 0.036,Y -516.838,Z 782.146,A 0.000,B 0.000,C 90.000,E1 242.281} C_DIS
LIN {X -0.154,Y -513.538,Z 782.136,A 0.000,B 0.000,C 90.000,E1 240.539} C_DIS
LIN {X -0.260,Y -510.723,Z 782.128,A 0.000,B 0.000,C 90.000,E1 239.076} C_DIS
LIN {X -0.049,Y -508.389,Z 782.122,A 0.000,B 0.000,C 90.000,E1 237.867} C_DIS
LIN {X 0.077,Y -506.581,Z 782.117,A 0.000,B 0.000,C 90.000,E1 236.962} C_DIS
LIN {X -0.201,Y -503.971,Z 782.110,A 0.000,B 0.000,C 90.000,E1 235.801} C_DIS
LIN {X -0.117,Y -501.956,Z 782.105,A 0.000,B 0.000,C 90.000,E1 234.895} C_DIS
LIN {X -0.059,Y -499.814,Z 782.100,A 0.000,B 0.000,C 90.000,E1 233.989} C_DIS
LIN {X 0.007,Y -496.061,Z 782.092,A 0.000,B 0.000,C 90.000,E1 232.477} C_DIS
LIN {X 0.012,Y -490.786,Z 782.080,A 0.000,B 0.000,C 90.000,E1 230.356} C_DIS
LIN {X -0.083,Y -483.811,Z 782.063,A 0.000,B 0.000,C 90.000,E1 227.310} C_DIS
LIN {X 0.260,Y -480.487,Z 782.054,A 0.000,B 0.000,C 90.000,E1 225.729} C_DIS
LIN {X 0.193,Y -477.106,Z 782.046,A 0.000,B 0.000,C 90.000,E1 224.190} C_DIS
LIN {X -0.169,Y -473.006,Z 782.035,A 0.000,B 0.000,C 90.000,E1 222.366} C_DIS
LIN {X 0.074,Y -468.924,Z 782.025,A 0.000,B 0.000,C 90.000,E1 220.458} C_DIS
LIN {X -0.086,Y -465.057,Z 782.014,A 0.000,B 0.000,C 90.000,E1 218.588} C_DIS
LIN {X -0.146,Y -460.346,Z 782.002,A 0.000,B 0.000,C 90.000,E1 216.377} C_DIS
LIN {X -0.062,Y -456.419,Z 781.991,A 0.000,B 0.000,C 90.000,E1 214.452} C_DIS
LIN {X -0.118,Y -451.852,Z 781.979,A 0.000,B 0.000,C 90.000,E1 212.212} C_DIS
LIN {X 0.012,Y -448.111,Z 781.968,A 0.000,B 0.000,C 90.000,E1 210.256} C_DIS
LIN {X 0.146,Y -444.978,Z 781.959,A 0.000,B 0.000,C 90.000,E1 208.615} C_DIS
LIN {X 0.009,Y -441.894,Z 781.950,A 0.000,B 0.000,C 90.000,E1 207.001} C_DIS
LIN {X 0.204,Y -438.754,Z 781.941,A 0.000,B 0.000,C 90.000,E1 205.335} C_DIS
LIN {X 0.145,Y -435.684,Z 781.932,A 0.000,B 0.000,C 90.000,E1 203.695} C_DIS
LIN {X -0.150,Y -432.545,Z 781.923,A 0.000,B 0.000,C 90.000,E1 202.078} C_DIS
LIN {X -0.072,Y -429.980,Z 781.915,A 0.000,B 0.000,C 90.000,E1 200.737} C_DIS
LIN {X 0.174,Y -425.475,Z 781.902,A 0.000,B 0.000,C 90.000,E1 198.362} C_DIS
LIN {X 0.190,Y -422.289,Z 781.893,A 0.000,B 0.000,C 90.000,E1 196.677} C_DIS
LIN {X -0.148,Y -419.644,Z 781.885,A 0.000,B 0.000,C 90.000,E1 195.371} C_DIS
LIN {X -0.134,Y -414.525,Z 781.870,A 0.000,B 0.000,C 90.000,E1 192.647} C_DIS
LIN {X 0.156,Y -411.375,Z 781.861,A 0.000,B 0.000,C 90.000,E1 190.894} C_DIS
LIN {X -0.012,Y -405.411,Z 781.841,A 0.000,B 0.000,C 90.000,E1 187.466} C_DIS
LIN {X -0.092,Y -402.460,Z 781.832,A 0.000,B 0.000,C 90.000,E1 185.739} C_DIS
LIN {X -0.183,Y -395.979,Z 781.808,A 0.000,B 0.000,C 90.000,E1 181.547} C_DIS
LIN {X 0.144,Y -393.019,Z 781.795,A 0.000,B 0.000,C 90.000,E1 179.026} C_DIS
LIN {X 0.019,Y -390.366,Z 781.781,A 0.000,B 0.000,C 90.000,E1 176.560} C_DIS
LIN {X 0.007,Y -388.670,Z 781.771,A 0.000,B 0.000,C 90.000,E1 174.780} C_DIS
LIN {X 0.170,Y -385.967,Z 781.755,A 0.000,B 0.000,C 90.000,E1 171.894} C_DIS
LIN {X -0.108,Y -383.355,Z 781.737,A 0.000,B 0.000,C 90.000,E1 168.701} C_DIS
LIN {X -0.170,Y -381.355,Z 781.719,A 0.000,B 0.000,C 90.000,E1 165.463} C_DIS
LIN {X -0.003,Y -380.321,Z 781.707,A 0.000,B 0.000,C 90.000,E1 163.268} C_DIS
LIN {X -0.014,Y -379.272,Z 781.689,A 0.000,B 0.000,C 90.000,E1 160.007} C_DIS
LIN {X 0.111,Y -378.858,Z 781.669,A 0.000,B 0.000,C 90.000,E1 156.357} C_DIS
LIN {X -0.135,Y -379.616,Z 781.651,A 0.000,B 0.000,C 90.000,E1 153.127} C_DIS
LIN {X -0.168,Y -381.723,Z 781.633,A 0.000,B 0.000,C 90.000,E1 149.871} C_DIS
LIN {X -0.017,Y -383.719,Z 781.622,A 0.000,B 0.000,C 90.000,E1 148.043} C_DIS
LIN {X 0.065,Y -388.043,Z 781.609,A 0.000,B 0.000,C 90.000,E1 145.515} C_DIS
LIN {X -0.042,Y -389.639,Z 781.605,A 0.000,B 0.000,C 90.000,E1 144.815} C_DIS
LIN {X 0.056,Y -392.310,Z 781.600,A 0.000,B 0.000,C 90.000,E1 143.909} C_DIS
LIN {X -0.019,Y -394.805,Z 781.596,A 0.000,B 0.000,C 90.000,E1 143.210} C_DIS
LIN {X -0.043,Y -396.999,Z 781.593,A 0.000,B 0.000,C 90.000,E1 142.683} C_DIS
LIN {X -0.082,Y -400.511,Z 781.589,A 0.000,B 0.000,C 90.000,E1 141.984} C_DIS
LIN {X -0.029,Y -404.195,Z 781.585,A 0.000,B 0.000,C 90.000,E1 141.376} C_DIS
LIN {X 0.261,Y -408.651,Z 781.582,A 0.000,B 0.000,C 90.000,E1 140.723} C_DIS
LIN {X 0.066,Y -427.430,Z 781.570,A 0.000,B 0.000,C 90.000,E1 138.528} C_DIS
LIN {X -0.081,Y -438.645,Z 781.563,A 0.000,B 0.000,C 90.000,E1 137.310} C_DIS
LIN {X 0.200,Y -449.649,Z 781.556,A 0.000,B 0.000,C 90.000,E1 136.053} C_DIS
LIN {X -0.144,Y -456.309,Z 781.552,A 0.000,B 0.000,C 90.000,E1 135.324} C_DIS
LIN {X 0.217,Y -460.066,Z 781.549,A 0.000,B 0.000,C 90.000,E1 134.838} C_DIS
LIN {X -0.220,Y -465.031,Z 781.546,A 0.000,B 0.000,C 90.000,E1 134.271} C_DIS
LIN {X 0.025,Y -473.631,Z 781.540,A 0.000,B 0.000,C 90.000,E1 133.137} C_DIS
LIN {X 0.110,Y -480.648,Z 781.535,A 0.000,B 0.000,C 90.000,E1 132.204} C_DIS
LIN {X -0.129,Y -486.159,Z 781.530,A 0.000,B 0.000,C 90.000,E1 131.472} C_DIS
LIN {X 0.157,Y -490.382,Z 781.527,A 0.000,B 0.000,C 90.000,E1 130.825} C_DIS
LIN {X 0.001,Y -496.506,Z 781.522,A 0.000,B 0.000,C 90.000,E1 129.930} C_DIS
LIN {X -0.184,Y -501.334,Z 781.518,A 0.000,B 0.000,C 90.000,E1 129.197} C_DIS
LIN {X 0.072,Y -508.435,Z 781.511,A 0.000,B 0.000,C 90.000,E1 127.971} C_DIS
LIN {X -0.002,Y -512.593,Z 781.507,A 0.000,B 0.000,C 90.000,E1 127.237} C_DIS
LIN {X -0.111,Y -518.086,Z 781.501,A 0.000,B 0.000,C 90.000,E1 126.217} C_DIS
LIN {X 0.091,Y -524.055,Z 781.495,A 0.000,B 0.000,C 90.000,E1 125.025} C_DIS
LIN {X -0.121,Y -526.197,Z 781.492,A 0.000,B 0.000,C 90.000,E1 124.612} C_DIS
LIN {X 0.040,Y -531.877,Z 781.485,A 0.000,B 0.000,C 90.000,E1 123.293} C_DIS
LIN {X -0.003,Y -537.074,Z 781.478,A 0.000,B 0.000,C 90.000,E1 122.005} C_DIS
LIN {X 0.166,Y -540.393,Z 781.473,A 0.000,B 0.000,C 90.000,E1 121.131} C_DIS
LIN {X 0.098,Y -543.431,Z 781.468,A 0.000,B 0.000,C 90.000,E1 120.285} C_DIS
LIN {X 0.087,Y -547.217,Z 781.462,A 0.000,B 0.000,C 90.000,E1 119.155} C_DIS
LIN {X 0.099,Y -549.918,Z 781.457,A 0.000,B 0.000,C 90.000,E1 118.309} C_DIS
LIN {X -0.088,Y -553.249,Z 781.451,A 0.000,B 0.000,C 90.000,E1 117.206} C_DIS
LIN {X -0.015,Y -555.330,Z 781.446,A 0.000,B 0.000,C 90.000,E1 116.360} C_DIS
LIN {X -0.167,Y -557.057,Z 781.442,A 0.000,B 0.000,C 90.000,E1 115.540} C_DIS
LIN {X -0.066,Y -558.525,Z 781.437,A 0.000,B 0.000,C 90.000,E1 114.695} C_DIS
LIN {X 0.322,Y -559.651,Z 781.433,A 0.000,B 0.000,C 90.000,E1 113.823} C_DIS
LIN {X -0.110,Y -561.498,Z 781.423,A 0.000,B 0.000,C 90.000,E1 112.206} C_DIS
LIN {X -0.101,Y -562.734,Z 781.417,A 0.000,B 0.000,C 90.000,E1 111.099} C_DIS
LIN {X -0.075,Y -563.774,Z 781.411,A 0.000,B 0.000,C 90.000,E1 109.993} C_DIS
LIN {X 0.096,Y -564.962,Z 781.403,A 0.000,B 0.000,C 90.000,E1 108.598} C_DIS
LIN {X -0.105,Y -566.200,Z 781.394,A 0.000,B 0.000,C 90.000,E1 106.968} C_DIS
LIN {X 0.261,Y -567.568,Z 781.384,A 0.000,B 0.000,C 90.000,E1 105.009} C_DIS
LIN {X 0.156,Y -569.325,Z 781.371,A 0.000,B 0.000,C 90.000,E1 102.827} C_DIS
LIN {X -0.217,Y -570.928,Z 781.361,A 0.000,B 0.000,C 90.000,E1 100.950} C_DIS
LIN {X 0.073,Y -572.065,Z 781.353,A 0.000,B 0.000,C 90.000,E1 99.557} C_DIS
LIN {X -0.068,Y -573.441,Z 781.344,A 0.000,B 0.000,C 90.000,E1 97.936} C_DIS
LIN {X -0.186,Y -574.578,Z 781.335,A 0.000,B 0.000,C 90.000,E1 96.315} C_DIS
LIN {X 0.028,Y -575.405,Z 781.327,A 0.000,B 0.000,C 90.000,E1 94.935} C_DIS
LIN {X -0.167,Y -576.338,Z 781.318,A 0.000,B 0.000,C 90.000,E1 93.326} C_DIS
LIN {X 0.047,Y -577.052,Z 781.311,A 0.000,B 0.000,C 90.000,E1 91.949} C_DIS
LIN {X 0.111,Y -577.552,Z 781.305,A 0.000,B 0.000,C 90.000,E1 90.859} C_DIS
LIN {X -0.090,Y -578.237,Z 781.296,A 0.000,B 0.000,C 90.000,E1 89.255} C_DIS
LIN {X -0.264,Y -578.808,Z 781.287,A 0.000,B 0.000,C 90.000,E1 87.650} C_DIS
LIN {X 0.144,Y -579.224,Z 781.278,A 0.000,B 0.000,C 90.000,E1 85.988} C_DIS
LIN {X 0.281,Y -579.477,Z 781.272,A 0.000,B 0.000,C 90.000,E1 84.894} C_DIS
LIN {X 0.214,Y -579.706,Z 781.263,A 0.000,B 0.000,C 90.000,E1 83.280} C_DIS
LIN {X 0.005,Y -579.959,Z 781.255,A 0.000,B 0.000,C 90.000,E1 81.951} C_DIS
LIN {X -0.207,Y -580.067,Z 781.248,A 0.000,B 0.000,C 90.000,E1 80.622} C_DIS
LIN {X 0.122,Y -580.157,Z 781.242,A 0.000,B 0.000,C 90.000,E1 79.511} C_DIS
LIN {X -0.224,Y -580.194,Z 781.236,A 0.000,B 0.000,C 90.000,E1 78.465} C_DIS
LIN {X -0.008,Y -580.022,Z 781.227,A 0.000,B 0.000,C 90.000,E1 76.825} C_DIS
LIN {X -0.009,Y -579.625,Z 781.216,A 0.000,B 0.000,C 90.000,E1 74.936} C_DIS
LIN {X 0.126,Y -579.110,Z 781.206,A 0.000,B 0.000,C 90.000,E1 73.032} C_DIS
LIN {X 0.211,Y -578.523,Z 781.197,A 0.000,B 0.000,C 90.000,E1 71.402} C_DIS
LIN {X 0.098,Y -577.859,Z 781.189,A 0.000,B 0.000,C 90.000,E1 70.061} C_DIS
LIN {X -0.024,Y -577.156,Z 781.182,A 0.000,B 0.000,C 90.000,E1 68.720} C_DIS
LIN {X 0.203,Y -576.505,Z 781.176,A 0.000,B 0.000,C 90.000,E1 67.614} C_DIS
LIN {X -0.271,Y -575.557,Z 781.168,A 0.000,B 0.000,C 90.000,E1 66.305} C_DIS
LIN {X -0.003,Y -574.456,Z 781.161,A 0.000,B 0.000,C 90.000,E1 64.921} C_DIS
LIN {X -0.117,Y -573.427,Z 781.155,A 0.000,B 0.000,C 90.000,E1 63.845} C_DIS
LIN {X 0.173,Y -572.517,Z 781.150,A 0.000,B 0.000,C 90.000,E1 62.999} C_DIS
LIN {X 0.126,Y -570.747,Z 781.143,A 0.000,B 0.000,C 90.000,E1 61.641} C_DIS
LIN {X -0.213,Y -570.001,Z 781.140,A 0.000,B 0.000,C 90.000,E1 61.129} C_DIS
LIN {X -0.037,Y -567.717,Z 781.132,A 0.000,B 0.000,C 90.000,E1 59.744} C_DIS
LIN {X -0.198,Y -565.673,Z 781.126,A 0.000,B 0.000,C 90.000,E1 58.663} C_DIS
LIN {X 0.092,Y -563.226,Z 781.120,A 0.000,B 0.000,C 90.000,E1 57.533} C_DIS
LIN {X -0.016,Y -561.940,Z 781.117,A 0.000,B 0.000,C 90.000,E1 56.993} C_DIS
LIN {X 0.046,Y -558.933,Z 781.111,A 0.000,B 0.000,C 90.000,E1 55.881} C_DIS
LIN {X 0.222,Y -557.364,Z 781.107,A 0.000,B 0.000,C 90.000,E1 55.308} C_DIS
LIN {X 0.147,Y -554.700,Z 781.103,A 0.000,B 0.000,C 90.000,E1 54.482} C_DIS
LIN {X 0.037,Y -551.828,Z 781.098,A 0.000,B 0.000,C 90.000,E1 53.657} C_DIS
LIN {X -0.277,Y -549.723,Z 781.095,A 0.000,B 0.000,C 90.000,E1 53.130} C_DIS
LIN {X -0.112,Y -546.224,Z 781.090,A 0.000,B 0.000,C 90.000,E1 52.271} C_DIS
LIN {X 0.159,Y -543.018,Z 781.086,A 0.000,B 0.000,C 90.000,E1 51.537} C_DIS
LIN {X -0.021,Y -539.526,Z 781.083,A 0.000,B 0.000,C 90.000,E1 50.848} C_DIS
LIN {X 0.011,Y -536.534,Z 781.079,A 0.000,B 0.000,C 90.000,E1 50.275} C_DIS
LIN {X 0.016,Y -533.209,Z 781.076,A 0.000,B 0.000,C 90.000,E1 49.703} C_DIS
LIN {X -0.064,Y -529.537,Z 781.073,A 0.000,B 0.000,C 90.000,E1 49.138} C_DIS
LIN {X -0.115,Y -525.442,Z 781.070,A 0.000,B 0.000,C 90.000,E1 48.566} C_DIS
LIN {X -0.120,Y -520.955,Z 781.067,A 0.000,B 0.000,C 90.000,E1 48.000} C_DIS
LIN {X -0.123,Y -514.928,Z 781.063,A 0.000,B 0.000,C 90.000,E1 47.310} C_DIS
LIN {X 0.009,Y -510.884,Z 781.060,A 0.000,B 0.000,C 90.000,E1 46.863} C_DIS
LIN {X 0.129,Y -505.239,Z 781.057,A 0.000,B 0.000,C 90.000,E1 46.296} C_DIS
LIN {X 0.203,Y -500.855,Z 781.055,A 0.000,B 0.000,C 90.000,E1 45.891} C_DIS
LIN {X 0.035,Y -494.761,Z 781.052,A 0.000,B 0.000,C 90.000,E1 45.405} C_DIS
LIN {X -0.006,Y -490.188,Z 781.050,A 0.000,B 0.000,C 90.000,E1 45.040} C_DIS
LIN {X -0.125,Y -480.832,Z 781.046,A 0.000,B 0.000,C 90.000,E1 44.352} C_DIS
LIN {X 0.101,Y -469.422,Z 781.042,A 0.000,B 0.000,C 90.000,E1 43.542} C_DIS
LIN {X -0.057,Y -456.452,Z 781.037,A 0.000,B 0.000,C 90.000,E1 42.690} C_DIS
LIN {X -0.028,Y -438.733,Z 781.030,A 0.000,B 0.000,C 90.000,E1 41.472} C_DIS
LIN {X -0.107,Y -416.891,Z 781.021,A 0.000,B 0.000,C 90.000,E1 39.850} C_DIS
LIN {X 0.099,Y -409.601,Z 781.018,A 0.000,B 0.000,C 90.000,E1 39.197} C_DIS
LIN {X 0.068,Y -407.192,Z 781.017,A 0.000,B 0.000,C 90.000,E1 38.955} C_DIS
LIN {X -0.190,Y -406.523,Z 781.016,A 0.000,B 0.000,C 90.000,E1 38.910} C_DIS
LIN {X -0.216,Y -406.497,Z 781.016,A 0.000,B 0.000,C 90.000,E1 38.910} C_DIS
LIN {X -0.054,Y -405.889,Z 781.014,A 0.000,B 0.000,C 90.000,E1 38.508} C_DIS
LIN {X 0.126,Y -397.279,Z 780.990,A 0.000,B 0.000,C 90.000,E1 34.119} C_DIS
LIN {X -0.212,Y -397.035,Z 780.989,A 0.000,B 0.000,C 90.000,E1 33.992} C_DIS
LIN {X 0.127,Y -397.871,Z 780.970,A 0.000,B 0.000,C 90.000,E1 30.590} C_DIS
LIN {X -0.034,Y -399.019,Z 780.956,A 0.000,B 0.000,C 90.000,E1 28.153} C_DIS
LIN {X 0.052,Y -400.627,Z 780.941,A 0.000,B 0.000,C 90.000,E1 25.335} C_DIS
LIN {X 0.020,Y -403.182,Z 780.921,A 0.000,B 0.000,C 90.000,E1 21.844} C_DIS
LIN {X -0.132,Y -407.361,Z 780.898,A 0.000,B 0.000,C 90.000,E1 17.692} C_DIS
LIN {X -0.058,Y -410.119,Z 780.887,A 0.000,B 0.000,C 90.000,E1 15.607} C_DIS
LIN {X 0.147,Y -414.317,Z 780.871,A 0.000,B 0.000,C 90.000,E1 12.827} C_DIS
LIN {X 0.165,Y -418.339,Z 780.858,A 0.000,B 0.000,C 90.000,E1 10.433} C_DIS
LIN {X 0.151,Y -421.866,Z 780.847,A 0.000,B 0.000,C 90.000,E1 8.398} C_DIS
LIN {X 0.066,Y -424.783,Z 780.837,A 0.000,B 0.000,C 90.000,E1 6.720} C_DIS
LIN {X 0.077,Y -428.363,Z 780.826,A 0.000,B 0.000,C 90.000,E1 4.702} C_DIS
LIN {X -0.069,Y -430.849,Z 780.819,A 0.000,B 0.000,C 90.000,E1 3.383} C_DIS
LIN {X 0.106,Y -435.337,Z 780.806,A 0.000,B 0.000,C 90.000,E1 1.031} C_DIS
LIN {X 0.162,Y -440.604,Z 780.792,A 0.000,B 0.000,C 90.000,E1 358.453} C_DIS
LIN {X 0.021,Y -447.226,Z 780.775,A 0.000,B 0.000,C 90.000,E1 355.527} C_DIS
LIN {X -0.052,Y -451.049,Z 780.766,A 0.000,B 0.000,C 90.000,E1 353.913} C_DIS
LIN {X 0.161,Y -455.629,Z 780.755,A 0.000,B 0.000,C 90.000,E1 351.951} C_DIS
LIN {X -0.144,Y -459.342,Z 780.747,A 0.000,B 0.000,C 90.000,E1 350.387} C_DIS
LIN {X 0.146,Y -462.903,Z 780.738,A 0.000,B 0.000,C 90.000,E1 348.757} C_DIS
LIN {X -0.014,Y -465.186,Z 780.732,A 0.000,B 0.000,C 90.000,E1 347.825} C_DIS
LIN {X 0.144,Y -467.023,Z 780.729,A 0.000,B 0.000,C 90.000,E1 347.173} C_DIS
LIN {X -0.241,Y -469.394,Z 780.725,A 0.000,B 0.000,C 90.000,E1 346.589} C_DIS
LIN {X -0.065,Y -471.409,Z 780.723,A 0.000,B 0.000,C 90.000,E1 346.172} C_DIS
LIN {X -0.049,Y -474.638,Z 780.721,A 0.000,B 0.000,C 90.000,E1 345.700} C_DIS
LIN {X -0.089,Y -477.830,Z 780.719,A 0.000,B 0.000,C 90.000,E1 345.338} C_DIS
LIN {X 0.019,Y -483.240,Z 780.716,A 0.000,B 0.000,C 90.000,E1 344.810} C_DIS
LIN {X -0.039,Y -493.384,Z 780.711,A 0.000,B 0.000,C 90.000,E1 344.031} C_DIS
LIN {X 0.185,Y -507.435,Z 780.706,A 0.000,B 0.000,C 90.000,E1 343.015} C_DIS
LIN {X -0.182,Y -523.247,Z 780.700,A 0.000,B 0.000,C 90.000,E1 342.000} C_DIS
LIN {X -0.050,Y -534.324,Z 780.696,A 0.000,B 0.000,C 90.000,E1 341.275} C_DIS
LIN {X 0.190,Y -542.077,Z 780.693,A 0.000,B 0.000,C 90.000,E1 340.732} C_DIS
LIN {X -0.239,Y -549.637,Z 780.690,A 0.000,B 0.000,C 90.000,E1 340.242} C_DIS
LIN {X -0.009,Y -553.856,Z 780.688,A 0.000,B 0.000,C 90.000,E1 339.880} C_DIS
LIN {X 0.056,Y -557.982,Z 780.686,A 0.000,B 0.000,C 90.000,E1 339.518} C_DIS
LIN {X -0.067,Y -563.338,Z 780.684,A 0.000,B 0.000,C 90.000,E1 339.028} C_DIS
LIN {X 0.327,Y -568.381,Z 780.681,A 0.000,B 0.000,C 90.000,E1 338.465} C_DIS
LIN {X -0.125,Y -573.182,Z 780.678,A 0.000,B 0.000,C 90.000,E1 337.975} C_DIS
LIN {X 0.073,Y -577.755,Z 780.675,A 0.000,B 0.000,C 90.000,E1 337.411} C_DIS
LIN {X 0.009,Y -583.024,Z 780.671,A 0.000,B 0.000,C 90.000,E1 336.741} C_DIS
LIN {X 0.159,Y -589.117,Z 780.666,A 0.000,B 0.000,C 90.000,E1 335.921} C_DIS
LIN {X 0.284,Y -596.553,Z 780.660,A 0.000,B 0.000,C 90.000,E1 334.845} C_DIS
LIN {X -0.025,Y -603.593,Z 780.655,A 0.000,B 0.000,C 90.000,E1 333.819} C_DIS
LIN {X 0.322,Y -609.382,Z 780.649,A 0.000,B 0.000,C 90.000,E1 332.871} C_DIS
LIN {X 0.191,Y -614.882,Z 780.644,A 0.000,B 0.000,C 90.000,E1 331.975} C_DIS
LIN {X 0.141,Y -617.922,Z 780.642,A 0.000,B 0.000,C 90.000,E1 331.463} C_DIS
LIN {X -0.145,Y -623.080,Z 780.637,A 0.000,B 0.000,C 90.000,E1 330.589} C_DIS
LIN {X 0.194,Y -629.465,Z 780.630,A 0.000,B 0.000,C 90.000,E1 329.410} C_DIS
LIN {X 0.039,Y -633.465,Z 780.626,A 0.000,B 0.000,C 90.000,E1 328.663} C_DIS
LIN {X -0.092,Y -636.600,Z 780.622,A 0.000,B 0.000,C 90.000,E1 328.043} C_DIS
